    slow_turning_mb:=H_SlowTurning OR BR_ECR_PUBSH_ALARM_TEST;    (*PRORCCAN1001	  slow_turning_mb      %QX284.0*)

       slow_turnok_mb:=SLOWTURNOK;      (*PRORCCAN1002	  slow_turnok_mb	      %QX284.1*)

       slow_turning_failure_mb:=SlowTurningFailure OR BR_ECR_PUBSH_ALARM_TEST ; (*PRORCCAN1003	low_turning_failure_mb	%QX284.2*)

	start_failure_alm:=startFail OR BR_ECR_PUBSH_ALARM_TEST;(*PRORCCAN1004   start_failure_alm   	%QX284.3*)

     start_air_valve_man_closed:=StartAirValueManClosedBX  OR BR_ECR_PUBSH_ALARM_TEST ;	(*PRORCCAN1005	start_air_valve_man_closed     %QX284.4*)

      turning_gear_engaged_alm:=H_TurnGearEngaged OR BR_ECR_PUBSH_ALARM_TEST;           (*PRORCCAN1006	turning_gear_engaged_alm	    %QX284.5-------------------------------------------*)

       turning_gear_sensor_failure_alm:=H_TurnGearSensorFail OR BR_ECR_PUBSH_ALARM_TEST;  (*PRORCCAN1007	turning_gear_sensor_failure_alm	%QX284.6 *)

       any_aux_blower_run_mb:=AnyAuxBlowerRun  OR BR_ECR_PUBSH_ALARM_TEST ;         (*PRORCCAN1008 	any_aux_blower_run_mb	      %QX284.7*)

       aux_blower_manctrl_mb:=H_AuxBlowerManCTRL;(*PRORCCAN1009	aux_blower_manctrl_mb  	%QX284.8*)

       aux_blower_failed_mb:=H_AuxBlowerFailed OR BR_ECR_PUBSH_ALARM_TEST;           (*PRORCCAN1010	aux_blower_failed_mb	       %QX284.9*)

       speed_prgm_override:=H_SPD_PRGM_OVERD;    (* PRORCCAN1011	speed_prgm_override   	       %QX284.10*)

       eng_output_limited:=H_ENG_OUTPUT_LIMITED;   (*PRORCCAN1012	eng_output_limited            	%QX284.11*)

       setpoint_critical_speed:=H_SETPOINT_CRITICAL_SPD_BX; (*PRORCCAN1013	setpoint_critical_speed    	%QX284.12 *)

       eng_critical_speed:=H_ENG_CRITICAL_SPD_BX;   (*PRORCCAN1014	eng_critical_speed     	%QX284.13*)

	unic_start_learning_inprogress_indica:= H_StartLearningInPro OR BR_ECR_PUBSH_ALARM_TEST; (*PRORCCAN1015	unic_start_learning_inprogress_indica  	%QX284.14*)

       speed_prgm_active:=H_SPEED_PRGM_ACTIVE;(*PRORCCAN1016   speed_prgm_active    %QX284.15*)

       bridge_ctrl:=BR_CTRL;(* PRORCCAN2001 	bridge_ctrl  	%QX285.0*)

        ecr_aut_ctrl:=ECRA_CTRL;  (*PRORCCAN2002	ecr_aut_ctrl  	%QX285.1*)

	 ecr_man_ctrl:=ECRM_CTRL;(*PRORCCAN2003	ecr_man_ctrl  	%QX285.2*)

	 local_man_ctrl:=LOC_MAN_CTRL;(*PRORCCAN2004 	local_man_ctrl  	%QX285.3*)

       br_lamp_br_flash:=BRG_BRG_CTRL_FLSH;      (*PRORCCAN2005	br_lamp_br_flash  	%QX285.4*)

	br_lamp_ecr_autom_flash:=BRG_ECRA_CTRL_FLSH;    (*PRORCCAN2006	br_lamp_ecr_autom_flash  	%QX285.5*)

	br_lamp_ecr_man_flash:=BRG_ECRM_CTRL_FLSH;   (*PRORCCAN2007	br_lamp_ecr_man_flash  	%QX285.6*)

	br_lamp_local_man_flash:=BRG_LOCAL_MAN_CTRL_FLSH;     (*PRORCCAN2008	br_lamp_local_man_flash  	%QX285.7*)

	br_accoustic_ctrl_transfer_signal:= BR_ACCOUST_CTRL_SIGN_BX;  (*PRORCCAN2009	br_accoustic_ctrl_transfer_signal  	%QX285.8*)

	ecr_lamp_br_flash:=ECR_BRG_CTRL_FLSH;   (*PRORCCAN2010	ecr_lamp_br_flash  	%QX285.9*)

	 ecr_lamp_ecr_autom_flash:=ECR_ECRA_CTRL_FLSH;(*PRORCCAN2011	ecr_lamp_ecr_autom_flash  	%QX285.10*)

	ecr_lamp_ecr_man_flash:=ECR_ECRM_CTRL_FLSH;(*PRORCCAN2012	ecr_lamp_ecr_man_flash   	%QX285.11*)

	ecr_lamp_local_man_flash:=ECR_LOCAL_MAN_CTRL_FLSH  ;(*PRORCCAN2013	ecr_lamp_local_man_flash   	%QX285.12*)

	ecr_ccoustic_ctrl_transfer_signal:= ECR_ACCOUST_CTRL_SIGN_BX ;  (*PRORCCAN2014	ecr_ccoustic_ctrl_transfer_signal  	%QX285.13*)

       shaft_locking_dev_engaged:= H_ShtLockDevEngaged OR BR_ECR_PUBSH_ALARM_TEST; (*PRORCCAN2015	  shaft_locking_dev_engaged     %QX285.14*)

       over_speed_rcs_mb:=OVER_SPEED;(*PRORCS0001   over_speed_rcs_mb	%QX286.0*)

	rcs_overspeed_sw:=RCS_SW_overspd;(*PRORCS0047	rcs_overspeed_sw  	%QX286.1*)

	rcs_overspeed_hw_mb:= RCS_HW_overspd; (*PRORCS0048	rcs_overspeed_hw_mb  	%QX286.2 *)

	air_run_indicator:=H_AIRRUN_BR_ECR;(*PRORCS0049	air_run_indicator  	%QX286.3*)

      rcs_mvl_br_failure:=MVL_BR_FAIL;(*PRORCS0050	rcs_mvl_br_failure  	%QX286.4*)

	rcs_mvl_ecr_failure:=MVL_ECR_FAIL;(*PRORCS0051	rcs_mvl_ecr_failure  	%QX286.5*)

       aux_blower_preselecRC_mb:=H_AuxBlowerPresel;(*PRORCS0052	aux_blower_preselecRC_mb	%QX286.6*)

	chief_limit_speed_indicaotr:=HMI_BR_ECRA_CHIEFLIMIT;  (*PRORCS0057	chief_limit_speed_indicaotr  	%QX286.7*)

       rcs_eng_speed_sensor1_failure:=RCS_SPD_SENSOR_FAIL1 OR BR_ECR_PUBSH_ALARM_TEST;    (*PRORCS0058	rcs_eng_speed_sensor1_failure	%QX286.8*)

	rcs_eng_speed_sensor2_failure:=RCS_SPD_SENSOR_FAIL2 OR BR_ECR_PUBSH_ALARM_TEST;  (*PRORCS0059	rcs_eng_speed_sensor2_failure	%QX286.9 *)

        startair_press_low_alm:=H_StartAirPressLow  OR BR_ECR_PUBSH_ALARM_TEST;  (*PRORCS0063	startair_press_low_alm   	%QX286.10----*)

       start_interlock_alm:= H_StartInterlock OR BR_ECR_PUBSH_ALARM_TEST 	;(*PRORCS0064	start_interlock_alm  	%QX286.11*)

       propulsion_ctrl_failure_alm_mb:=propulsion_ctrl_failure_alm;  (*PRORCS0069 	propulsion_ctrl_failure_alm   	%QX286.12*)

       propulsion_ctrl_passive_failure_alm_mb:=propulsion_ctrl_passive_failure_alm;(*  PRORCS0070  propulsion_ctrl_passive_failure_alm_mb  %QX286.13*)

	propulsion_ctrl_speed_meas_failure_alm:=PCS_SPD_MEASURE_FAILURE; (*PRORCS0071	propulsion_ctrl_speed_meas_failure_alm  	%QX286.14*)

       rcs_comm_to_unic_lost_failure:=CommunicationLost OR BR_ECR_PUBSH_ALARM_TEST;	(* PRORCS0072	rcs_comm_to_unic_lost_failure  	%QX287.0*)

       rcs_can1_TO_unic_lost_failure:=BreakDownCAN1 OR  BR_ECR_PUBSH_ALARM_TEST;	(*PRORCS0073	rcs_can1_TO_unic_lost_failure  	%QX287.1*)

       rcs_can2_to_unic_lost_failure:=BreakDownCAN2 OR  BR_ECR_PUBSH_ALARM_TEST ;  	(*PRORCS0074	rcs_can2_TO_unic_lost_failure  	%QX287.2*)

	eng_starting:= START AND (EngTurnINCRSPDir AND  NOT EngineStandstill )  OR BR_ECR_PUBSH_ALARM_TEST; (*PRORCS0075	eng_starting  	%QX287.3*)

	eng_running:=EngineRun OR BR_ECR_PUBSH_ALARM_TEST; (*PRORCS0076	eng_running  	%QX287.4*)

	eng_ready_for_start:= NOT  eng_not_ready OR BR_ECR_PUBSH_ALARM_TEST; (*PRORCS0077	eng_ready_for_start  	%QX287.5*)

	eng_not_ready:=StartInterlock  OR CommunicationLost  OR BR_ECR_PUBSH_ALARM_TEST ;(*PRORCS0078	eng_not_ready  	%QX287.6*)

	eng_stopping:=( NOT NNBrake AND  BRAKE  ) OR BR_ECR_PUBSH_ALARM_TEST; (*PRORCS0079 	eng_stopping  	%QX287.7*)

	eng_stopped:=EngineStandstill;(*PRORCS0080	eng_stopped  	%QX287.8*)

	rcs_eng_speed2:=ANALOG_DETECT_SPEED_RCS;(*PRORCS0081	rcs_eng_speed2	%QX300*)

	safety_system_off:= SafetySystemOff  OR BR_ECR_PUBSH_ALARM_TEST;  (*PRORCS0082	safety_system_off  	%QX287.10*)

	eng_tripped_mb:=eng_tripped OR BR_ECR_PUBSH_ALARM_TEST;   (*eng_tripped_mb  AT  %QX266.11:BOOL  ;*)(*PRORCS0083	eng_tripped  	%QX287.11*)

	mvl_postion_ahead  :=MVL_POS_AHD  ;(*PRORCS0091	mvl_postion_ahead  	%QX287.12*)

	mvl_postion_astern :=MVL_POS_AST ;(*PRORCS0092	mvl_postion_astern  	%QX287.13*)

	mvl_postion_stop  :=MVL_POS_STOP;(*PRORCS0093	mvl_postion_stop  	%QX287.14*)

	ahead_cmd:=AHEAD;   (*PRORCS0094	ahead_cmd  	%QX288.0*)

	 astern_cmd:=   ASTERN;    (*PRORCS0095	astern_cmd  	%QX288.1*)

	stop_cmd:=STOP;   (*PRORCS0096	stop_cmd  	%QX288.2*)

       rcs_eng_turning_ahead :=EngTurningAHD; (*PRORCS0099	rcs_eng_turning_ahead  	%QX288.3*)

	rcs_eng_turning_astern := EngTurningAST ; (*PRORCS0100	rcs_eng_turning_astern   	%QX288.4*)

       pcs_system_ready:= RemoteCtrl AND NOT (CommunicationLost  OR ess_can_communicationLost  OR  propulsion_ctrl_failure_alm OR  SafetySystemOff) OR BR_ECR_PUBSH_ALARM_TEST ;(*PRORCS0103	pcs_system_ready  	%QX288.5    ALARM  TEST*)

       plant_interlock:=PlantInterlock;(*PRORCS0107	plant_interlock  	%QX288.6*)

        remote_ctrl_failure:=propulsion_ctrl_failure_alm  OR BR_ECR_PUBSH_ALARM_TEST; (*PRORCS0108	remote_ctrl_failure  	%QX288.7 *)

	(* wrong_way_alm:=H_WRONG_WAY_ALARM;(*PRORCS0109	wrong_way_alm  	%QX288.8*)--------------DELETE*)

        ecr_lamp_test_pb_mb:=ECR_LAMP_TEST_PB_INTERNAL;(*PRORCS0139	ecr_lamp_test_pb_mb	%QX288.9*)

        br_lamp_test_pb_mb:=BR_LAMP_TEST_PB_INTERNAL;(*PRORCS0140	br_lamp_test_pb_mb	%QX288.10*)

	  br_portlamp_test_pb_mb:=BR_LAMP_TEST_PB_INTERNAL;(*PRORCS0141	br_portlamp_test_pb_mb	%QX288.11*)

	 br_stbdlamp_test_pb_mb:=BR_LAMP_TEST_PB_INTERNAL;(*PRORCS0142	br_stbdlamp_test_pb_mb	%QX288.12 *)

       spd_sim_mode_active_mb:=SPD_SIM_MODE_ACTIVE_FLAG;(* PRORCS0157	spd_sim_mode_active_mb	%QX289.11*)

	 startfail_horn_alm_mb:=Start_Fail_Flash_sign;   (*PRORCS0158   	StartFail HORN ALARM		SP_swd_perm_rcs6_13_62 	*)

      (* horn_alarm_mb:=(H_HORN_ALARM_ECR OR H_HORN_ALARM_BRG  OR ENG_FAIL_ACOUSTIC OR BR_ECR_PUBSH_ALARM_TEST) ; *)(*PRORCS0164	horn_alarm_mb	%QX289.13*)


        port_ctrl_rc_es:= PORT_CTRL_EOT ;(*PRORCS9001	port_ctrl_rc_es	%QX287.9*)

        stbd_ctrl_rc_es:=STBD_CTRL_EOT ;(*PRORCS9002	stbd   ctrl_rc_es*)

        rcs_speed_meansure_value_mb:=RCS_SPEED_MEANSURE_VALUE;(*PRORCS9003	rcs_speed_meansure_value_mb	%QX302*)

        safety_sys_stop_mb:=  SafetyStop;(*PRORCS9004*)

        br_mvl_level_mb:=BR_MVL_LEVEL;(*%QW370*)

        ecr_mvl_level_mb:=ECR_MVL_LEVEL;(*%QW372*)

       br_ecr_pubsh_alarm_test_mb:=BR_ECR_PUBSH_ALARM_TEST;

	h_br_mvl_rpm_cmd_mb:=BR_MVL_RPM_CMD ;(*%QW468*)

	h_ecr_mvl_rpm_cmd_mb:=MCR_MVL_RPM_CMD;(*%QW470*)
END_FUNCTION_BLOCK

(* POU Configuration/MODBUS_CONFIGURATION, ST *)
PROGRAM MODBUS_CONFIGURATION        
VAR                                
END_VAR                            
(*                                 
   <?xml version="1.0" encoding="UTF-16" standalone="yes"?>
<network xml_structure_version="1">
	<generator_settings minRTUTaskCycleTimeMs="5" minEthaskCycleTimeMs="5" ethSlaveMultiplier="0.1" rtuInterfaceMultiplier="0.1" taskGeneration="false"/>
	<master_interface type="eth" name="" expanded="true">
		<mb_slave comment="Ethernet MR Controller 100MBit 2Port" name="ESS" expanded="false" type="wago" article-no="0750-0882">
			<mb_connection type="eth" transport="UDP" port="502" ip="192.168.1.2" unitid="2" request_delay_ms="0" response_timeout_ms="50"/>
			<service_connection type="eth" ip="192.168.1.2"/>
			<generic_vars comment="" expanded="false"/>
			<pfc_vars comment="" expanded="true">
				<pfc_var name="ess_eng_turning_ahead_bkp_cfg" comment="" data_type="BOOL" iec_addr="%QX272.0" expanded="false" mb_access="ro" explicitAccess="false"/>
				<pfc_var name="ess_eng_turning_astern_bkp_cfg" comment="" data_type="BOOL" iec_addr="%QX272.1" expanded="false" mb_access="ro" explicitAccess="false"/>
				<pfc_var name="ess_eng_standstill_bkp_cfg" comment="" data_type="BOOL" iec_addr="%QX270.0" expanded="false" mb_access="ro" explicitAccess="false"/>
				<pfc_var name="ess_overspeed_sw_bkp_cfg" comment="" data_type="BOOL" iec_addr="%QX271.11" expanded="false" mb_access="ro" explicitAccess="false"/>
				<pfc_var name="ess_overspeed_hw_bkp_cfg" comment="" data_type="BOOL" iec_addr="%QX272.2" expanded="false" mb_access="ro" explicitAccess="false"/>
				<pfc_var name="alrm_acksound_off_br_cfg" comment="" data_type="BOOL" iec_addr="%QX274.1" expanded="false" mb_access="ro" explicitAccess="false"/>
				<pfc_var name="alrm_acksound_off_ecr_cfg" comment="" data_type="BOOL" iec_addr="%QX274.2" expanded="false" mb_access="ro" explicitAccess="false"/>
				<pfc_var name="alrm_acksound_off_port_cfg" comment="" data_type="BOOL" iec_addr="%QX274.3" expanded="false" mb_access="ro" explicitAccess="false"/>
				<pfc_var name="alrm_acksound_off_stbd_cfg" comment="" data_type="BOOL" iec_addr="%QX274.4" expanded="false" mb_access="ro" explicitAccess="false"/>
				<pfc_var name="safety_stop_cfg" comment="" data_type="BOOL" iec_addr="%QX271.13" expanded="false" mb_access="ro" explicitAccess="false"/>
				<pfc_var name="ess_eng_speed_bkp_cfg" comment="" data_type="REAL" iec_addr="%QW256" expanded="false" mb_access="ro" explicitAccess="false"/>
				<pfc_var name="ess_can_communicationLost_cfg" comment="" data_type="BOOL" iec_addr="%QX270.7" expanded="false" mb_access="ro" explicitAccess="false"/>
			</pfc_vars>
			<k_bus comment="" expanded="false"/>
		</mb_slave>
		<mb_slave comment="Ethernet MR Controller 100MBit 2Port" name="EOT" expanded="false" type="wago" article-no="0750-0882">
			<mb_connection type="eth" transport="UDP" port="502" ip="192.168.1.3" unitid="3" request_delay_ms="0" response_timeout_ms="50"/>
			<service_connection type="eth" ip="192.168.1.3"/>
			<generic_vars comment="" expanded="false"/>
			<pfc_vars comment="" expanded="true">
				<pfc_var name="BR_MVL_cfg" comment="" data_type="WORD" iec_addr="%QW0" expanded="false" mb_access="ro" explicitAccess="false"/>
				<pfc_var name="ECR_MVL_cfg" comment="" data_type="WORD" iec_addr="%QW1" expanded="false" mb_access="ro" explicitAccess="false"/>
			</pfc_vars>
			<k_bus comment="" expanded="false"/>
		</mb_slave>
		<mb_slave comment="Ethernet MR Controller 100MBit 2Port" name="ESS_2" expanded="true" type="wago" article-no="0750-0882">
			<mb_connection type="eth" transport="UDP" port="502" ip="192.168.2.2" unitid="2" request_delay_ms="0" response_timeout_ms="50"/>
			<service_connection type="eth" ip="192.168.1.2"/>
			<generic_vars comment="" expanded="false"/>
			<pfc_vars comment="" expanded="true">
				<pfc_var name="ess_eng_turning_ahead_bkp_cfg" comment="" data_type="BOOL" iec_addr="%QX272.0" expanded="false" mb_access="ro" explicitAccess="false"/>
				<pfc_var name="ess_eng_turning_astern_bkp_cfg" comment="" data_type="BOOL" iec_addr="%QX272.1" expanded="false" mb_access="ro" explicitAccess="false"/>
				<pfc_var name="ess_eng_standstill_bkp_cfg" comment="" data_type="BOOL" iec_addr="%QX270.0" expanded="false" mb_access="ro" explicitAccess="false"/>
				<pfc_var name="ess_overspeed_sw_bkp_cfg" comment="" data_type="BOOL" iec_addr="%QX271.11" expanded="false" mb_access="ro" explicitAccess="false"/>
				<pfc_var name="ess_overspeed_hw_bkp_cfg" comment="" data_type="BOOL" iec_addr="%QX272.2" expanded="false" mb_access="ro" explicitAccess="false"/>
				<pfc_var name="alrm_acksound_off_br_cfg" comment="" data_type="BOOL" iec_addr="%QX274.1" expanded="false" mb_access="ro" explicitAccess="false"/>
				<pfc_var name="alrm_acksound_off_ecr_cfg" comment="" data_type="BOOL" iec_addr="%QX274.2" expanded="false" mb_access="ro" explicitAccess="false"/>
				<pfc_var name="alrm_acksound_off_port_cfg" comment="" data_type="BOOL" iec_addr="%QX274.3" expanded="false" mb_access="ro" explicitAccess="false"/>
				<pfc_var name="alrm_acksound_off_stbd_cfg" comment="" data_type="BOOL" iec_addr="%QX274.4" expanded="false" mb_access="ro" explicitAccess="false"/>
				<pfc_var name="safety_stop_cfg" comment="" data_type="BOOL" iec_addr="%QX271.13" expanded="false" mb_access="ro" explicitAccess="false"/>
				<pfc_var name="ess_eng_speed_bkp_cfg" comment="" data_type="REAL" iec_addr="%QW256" expanded="false" mb_access="ro" explicitAccess="false"/>
				<pfc_var name="ess_can_communicationLost_cfg" comment="" data_type="BOOL" iec_addr="%QX270.7" expanded="false" mb_access="ro" explicitAccess="false"/>
			</pfc_vars>
			<k_bus comment="" expanded="false"/>
		</mb_slave>
	</master_interface>
</network>
                              
*)                                 
;                                  
END_PROGRAM

(* POU Generated Code/Ethernet/MBCFG_ESS, ST *)
PROGRAM MBCFG_ESS(* generated by config one prg for each slave *)

VAR_INPUT

END_VAR

VAR_OUTPUT
       ess_eng_turning_ahead_bkp_cfg       :    BOOL;       (**) 
       ess_eng_turning_astern_bkp_cfg       :    BOOL;       (**) 
       ess_eng_standstill_bkp_cfg       :    BOOL;       (**) 
       ess_overspeed_sw_bkp_cfg       :    BOOL;       (**) 
       ess_overspeed_hw_bkp_cfg       :    BOOL;       (**) 
       alrm_acksound_off_br_cfg       :    BOOL;       (**) 
       alrm_acksound_off_ecr_cfg       :    BOOL;       (**) 
       alrm_acksound_off_port_cfg       :    BOOL;       (**) 
       alrm_acksound_off_stbd_cfg       :    BOOL;       (**) 
       safety_stop_cfg       :    BOOL;       (**) 
       ess_eng_speed_bkp_cfg       :    REAL;       (**) 
       ess_can_communicationLost_cfg       :    BOOL;       (**) 

    (*--- system variables (read only) ----------------------------------------*)
    MBCFG_IpAddress :   STRING(11) := '192.168.1.2'; (* address of this slave *)
    MBCFG_Port      :   UINT := 502;
    MBCFG_UnitID    :   BYTE := 2;
    MBCFG_TimeOut   :   TIME := t#50ms;
    MBCFG_Error     :   MBCFG_eERROR;
    (*-------------------------------------------------------------------------*)
END_VAR

{library private}
VAR CONSTANT
    zz_VARIABLECOUNT:   INT := 12;	(* number of variables 	*)
    zz_JOBCOUNT     :   INT := 2; 	(* number of jobs		*)
END_VAR
VAR

    (*=== VARIABLE LIST ===============================================================================*)
    zz_VariableList :   ARRAY[1..zz_VARIABLECOUNT] OF MBCFG_typVARIABLE :=
    (   BitSize         := 1,
        ptVar           := 0,
        ReadJobIndex    := 1,
        ReadStartBitNo  := 32,
        WriteJobIndex   := 0,
        WriteStartBitNo := 0 ),
    (   BitSize         := 1,
        ptVar           := 0,
        ReadJobIndex    := 1,
        ReadStartBitNo  := 33,
        WriteJobIndex   := 0,
        WriteStartBitNo := 0 ),
    (   BitSize         := 1,
        ptVar           := 0,
        ReadJobIndex    := 1,
        ReadStartBitNo  := 0,
        WriteJobIndex   := 0,
        WriteStartBitNo := 0 ),
    (   BitSize         := 1,
        ptVar           := 0,
        ReadJobIndex    := 1,
        ReadStartBitNo  := 27,
        WriteJobIndex   := 0,
        WriteStartBitNo := 0 ),
    (   BitSize         := 1,
        ptVar           := 0,
        ReadJobIndex    := 1,
        ReadStartBitNo  := 34,
        WriteJobIndex   := 0,
        WriteStartBitNo := 0 ),
    (   BitSize         := 1,
        ptVar           := 0,
        ReadJobIndex    := 1,
        ReadStartBitNo  := 65,
        WriteJobIndex   := 0,
        WriteStartBitNo := 0 ),
    (   BitSize         := 1,
        ptVar           := 0,
        ReadJobIndex    := 1,
        ReadStartBitNo  := 66,
        WriteJobIndex   := 0,
        WriteStartBitNo := 0 ),
    (   BitSize         := 1,
        ptVar           := 0,
        ReadJobIndex    := 1,
        ReadStartBitNo  := 67,
        WriteJobIndex   := 0,
        WriteStartBitNo := 0 ),
    (   BitSize         := 1,
        ptVar           := 0,
        ReadJobIndex    := 1,
        ReadStartBitNo  := 68,
        WriteJobIndex   := 0,
        WriteStartBitNo := 0 ),
    (   BitSize         := 1,
        ptVar           := 0,
        ReadJobIndex    := 1,
        ReadStartBitNo  := 29,
        WriteJobIndex   := 0,
        WriteStartBitNo := 0 ),
    (   BitSize         := 32,
        ptVar           := 0,
        ReadJobIndex    := 2,
        ReadStartBitNo  := 0,
        WriteJobIndex   := 0,
        WriteStartBitNo := 0 ),
    (   BitSize         := 1,
        ptVar           := 0,
        ReadJobIndex    := 1,
        ReadStartBitNo  := 7,
        WriteJobIndex   := 0,
        WriteStartBitNo := 0 )

                        ;
    (*=================================================================================================*)

    (*=== JOB LIST ====================================================================================*)
    zz_JobList     :   ARRAY[1..zz_JOBCOUNT] OF MBCFG_typCOM_JOB :=
     (   Functioncode            := 2,
        ReadStartAddress        := 4320,
        ReadQuantity            := 69,
        WriteStartAddress       := 0,
        WriteQuantity           := 0,
        ptReadData              := 0, 
        ptWriteData             := 0 ),
     (   Functioncode            := 4,
        ReadStartAddress        := 256,
        ReadQuantity            := 2,
        WriteStartAddress       := 0,
        WriteQuantity           := 0,
        ptReadData              := 0, 
        ptWriteData             := 0 )

                        ;
    (*=================================================================================================*)

    (*=== DATA FIELDS =================================================================================*)
     zz_DataField_1_Read       :       ARRAY[1..5] OF WORD;
     zz_DataField_2_Read       :       ARRAY[1..2] OF WORD;
	
    (*=================================================================================================*)

    (*=== MODBUS MASTER =====================================*)
    zz_MBCFG_MASTER_ETH :       MBCFG_MASTER_UDP;
    (*=======================================================*)

END_VAR
(*--- for each variable -------------------------*)
   zz_VariableList[1].ptVar := ADR(ess_eng_turning_ahead_bkp_cfg);
   zz_VariableList[2].ptVar := ADR(ess_eng_turning_astern_bkp_cfg);
   zz_VariableList[3].ptVar := ADR(ess_eng_standstill_bkp_cfg);
   zz_VariableList[4].ptVar := ADR(ess_overspeed_sw_bkp_cfg);
   zz_VariableList[5].ptVar := ADR(ess_overspeed_hw_bkp_cfg);
   zz_VariableList[6].ptVar := ADR(alrm_acksound_off_br_cfg);
   zz_VariableList[7].ptVar := ADR(alrm_acksound_off_ecr_cfg);
   zz_VariableList[8].ptVar := ADR(alrm_acksound_off_port_cfg);
   zz_VariableList[9].ptVar := ADR(alrm_acksound_off_stbd_cfg);
   zz_VariableList[10].ptVar := ADR(safety_stop_cfg);
   zz_VariableList[11].ptVar := ADR(ess_eng_speed_bkp_cfg);
   zz_VariableList[12].ptVar := ADR(ess_can_communicationLost_cfg);

(*-----------------------------------------------*)

(*--- for each job -----------------------------------*)
zz_JobList[1].ptReadData   := ADR(zz_DataField_1_Read);
zz_JobList[2].ptReadData   := ADR(zz_DataField_2_Read);

(*----------------------------------------------------*)


(*#### START OF FIXED CODE #####################################*)
zz_MBCFG_MASTER_ETH(	strIpAddress    := MBCFG_IpAddress,
                        uiPort          := MBCFG_Port,
                        bUnitID         := MBCFG_UnitID,
                        tTimeOut        := MBCFG_TimeOut,
                        iVariableCount  := zz_VARIABLECOUNT,
                        ptVariableList  := ADR(zz_VariableList),
                        iJobCount       := zz_JOBCOUNT,
                        ptJobList       := ADR(zz_JobList),
                        eError          => MBCFG_Error
                    );
(*##############################################################*)
END_PROGRAM

(* POU Generated Code/Ethernet/MBCFG_ESS_2, ST *)
PROGRAM MBCFG_ESS_2(* generated by config one prg for each slave *)

VAR_INPUT

END_VAR

VAR_OUTPUT
       ess_eng_turning_ahead_bkp_cfg       :    BOOL;       (**) 
       ess_eng_turning_astern_bkp_cfg       :    BOOL;       (**) 
       ess_eng_standstill_bkp_cfg       :    BOOL;       (**) 
       ess_overspeed_sw_bkp_cfg       :    BOOL;       (**) 
       ess_overspeed_hw_bkp_cfg       :    BOOL;       (**) 
       alrm_acksound_off_br_cfg       :    BOOL;       (**) 
       alrm_acksound_off_ecr_cfg       :    BOOL;       (**) 
       alrm_acksound_off_port_cfg       :    BOOL;       (**) 
       alrm_acksound_off_stbd_cfg       :    BOOL;       (**) 
       safety_stop_cfg       :    BOOL;       (**) 
       ess_eng_speed_bkp_cfg       :    REAL;       (**) 
       ess_can_communicationLost_cfg       :    BOOL;       (**) 

    (*--- system variables (read only) ----------------------------------------*)
    MBCFG_IpAddress :   STRING(11) := '192.168.2.2'; (* address of this slave *)
    MBCFG_Port      :   UINT := 502;
    MBCFG_UnitID    :   BYTE := 2;
    MBCFG_TimeOut   :   TIME := t#50ms;
    MBCFG_Error     :   MBCFG_eERROR;
    (*-------------------------------------------------------------------------*)
END_VAR

{library private}
VAR CONSTANT
    zz_VARIABLECOUNT:   INT := 12;	(* number of variables 	*)
    zz_JOBCOUNT     :   INT := 2; 	(* number of jobs		*)
END_VAR
VAR

    (*=== VARIABLE LIST ===============================================================================*)
    zz_VariableList :   ARRAY[1..zz_VARIABLECOUNT] OF MBCFG_typVARIABLE :=
    (   BitSize         := 1,
        ptVar           := 0,
        ReadJobIndex    := 1,
        ReadStartBitNo  := 32,
        WriteJobIndex   := 0,
        WriteStartBitNo := 0 ),
    (   BitSize         := 1,
        ptVar           := 0,
        ReadJobIndex    := 1,
        ReadStartBitNo  := 33,
        WriteJobIndex   := 0,
        WriteStartBitNo := 0 ),
    (   BitSize         := 1,
        ptVar           := 0,
        ReadJobIndex    := 1,
        ReadStartBitNo  := 0,
        WriteJobIndex   := 0,
        WriteStartBitNo := 0 ),
    (   BitSize         := 1,
        ptVar           := 0,
        ReadJobIndex    := 1,
        ReadStartBitNo  := 27,
        WriteJobIndex   := 0,
        WriteStartBitNo := 0 ),
    (   BitSize         := 1,
        ptVar           := 0,
        ReadJobIndex    := 1,
        ReadStartBitNo  := 34,
        WriteJobIndex   := 0,
        WriteStartBitNo := 0 ),
    (   BitSize         := 1,
        ptVar           := 0,
        ReadJobIndex    := 1,
        ReadStartBitNo  := 65,
        WriteJobIndex   := 0,
        WriteStartBitNo := 0 ),
    (   BitSize         := 1,
        ptVar           := 0,
        ReadJobIndex    := 1,
        ReadStartBitNo  := 66,
        WriteJobIndex   := 0,
        WriteStartBitNo := 0 ),
    (   BitSize         := 1,
        ptVar           := 0,
        ReadJobIndex    := 1,
        ReadStartBitNo  := 67,
        WriteJobIndex   := 0,
        WriteStartBitNo := 0 ),
    (   BitSize         := 1,
        ptVar           := 0,
        ReadJobIndex    := 1,
        ReadStartBitNo  := 68,
        WriteJobIndex   := 0,
        WriteStartBitNo := 0 ),
    (   BitSize         := 1,
        ptVar           := 0,
        ReadJobIndex    := 1,
        ReadStartBitNo  := 29,
        WriteJobIndex   := 0,
        WriteStartBitNo := 0 ),
    (   BitSize         := 32,
        ptVar           := 0,
        ReadJobIndex    := 2,
        ReadStartBitNo  := 0,
        WriteJobIndex   := 0,
        WriteStartBitNo := 0 ),
    (   BitSize         := 1,
        ptVar           := 0,
        ReadJobIndex    := 1,
        ReadStartBitNo  := 7,
        WriteJobIndex   := 0,
        WriteStartBitNo := 0 )

                        ;
    (*=================================================================================================*)

    (*=== JOB LIST ====================================================================================*)
    zz_JobList     :   ARRAY[1..zz_JOBCOUNT] OF MBCFG_typCOM_JOB :=
     (   Functioncode            := 2,
        ReadStartAddress        := 4320,
        ReadQuantity            := 69,
        WriteStartAddress       := 0,
        WriteQuantity           := 0,
        ptReadData              := 0, 
        ptWriteData             := 0 ),
     (   Functioncode            := 4,
        ReadStartAddress        := 256,
        ReadQuantity            := 2,
        WriteStartAddress       := 0,
        WriteQuantity           := 0,
        ptReadData              := 0, 
        ptWriteData             := 0 )

                        ;
    (*=================================================================================================*)

    (*=== DATA FIELDS =================================================================================*)
     zz_DataField_1_Read       :       ARRAY[1..5] OF WORD;
     zz_DataField_2_Read       :       ARRAY[1..2] OF WORD;
	
    (*=================================================================================================*)

    (*=== MODBUS MASTER =====================================*)
    zz_MBCFG_MASTER_ETH :       MBCFG_MASTER_UDP;
    (*=======================================================*)

END_VAR
(*--- for each variable -------------------------*)
   zz_VariableList[1].ptVar := ADR(ess_eng_turning_ahead_bkp_cfg);
   zz_VariableList[2].ptVar := ADR(ess_eng_turning_astern_bkp_cfg);
   zz_VariableList[3].ptVar := ADR(ess_eng_standstill_bkp_cfg);
   zz_VariableList[4].ptVar := ADR(ess_overspeed_sw_bkp_cfg);
   zz_VariableList[5].ptVar := ADR(ess_overspeed_hw_bkp_cfg);
   zz_VariableList[6].ptVar := ADR(alrm_acksound_off_br_cfg);
   zz_VariableList[7].ptVar := ADR(alrm_acksound_off_ecr_cfg);
   zz_VariableList[8].ptVar := ADR(alrm_acksound_off_port_cfg);
   zz_VariableList[9].ptVar := ADR(alrm_acksound_off_stbd_cfg);
   zz_VariableList[10].ptVar := ADR(safety_stop_cfg);
   zz_VariableList[11].ptVar := ADR(ess_eng_speed_bkp_cfg);
   zz_VariableList[12].ptVar := ADR(ess_can_communicationLost_cfg);

(*-----------------------------------------------*)

(*--- for each job -----------------------------------*)
zz_JobList[1].ptReadData   := ADR(zz_DataField_1_Read);
zz_JobList[2].ptReadData   := ADR(zz_DataField_2_Read);

(*----------------------------------------------------*)


(*#### START OF FIXED CODE #####################################*)
zz_MBCFG_MASTER_ETH(	strIpAddress    := MBCFG_IpAddress,
                        uiPort          := MBCFG_Port,
                        bUnitID         := MBCFG_UnitID,
                        tTimeOut        := MBCFG_TimeOut,
                        iVariableCount  := zz_VARIABLECOUNT,
                        ptVariableList  := ADR(zz_VariableList),
                        iJobCount       := zz_JOBCOUNT,
                        ptJobList       := ADR(zz_JobList),
                        eError          => MBCFG_Error
                    );
(*##############################################################*)
END_PROGRAM

(* POU SWD, ST *)
FUNCTION_BLOCK SWD
VAR_INPUT
END_VAR
VAR_OUTPUT
END_VAR
VAR
	SRinst:SR;
	AIR_RUN_START_TEMP:BOOL;
	AIR_RUN_STOP_TEMP:BOOL;
	TOFInst_wgf: TOF;
	Slow_turning_staible:BOOL;
END_VAR
(*----------------SWD_swd_me_62   PROSWD0001----------------------*)
(*
IF   startFail   THEN   SWD_swd_me_62:=8;(*me_start_failure  8*)

ELSIF  ( NOT NNBrake)  AND  BRAKE    THEN  SWD_swd_me_62:=4 ;(* Stoping* ----------------ENG BRAKING???-------*)
(*ELSIF  (STOP AND EngineStandstill=FALSE)   THEN   SWD_swd_me_62:=4;(*me_stopping  4  *)*)
ELSIF   EngineRun    THEN   SWD_swd_me_62:=1;(* me_running    1 *)

ELSIF    EngineStandstill AND (NOT eng_ready_for_start)  THEN   SWD_swd_me_62:=3;(* me_stopped   3 *)
ELSIF    StartInterlock   THEN   SWD_swd_me_62:=2;(* me_startinterlock  2  *)
ELSIF   SlowTurningBX   THEN   SWD_swd_me_62:=6;(* me_slow_turning  6 *)
ELSIF   (PRESTART  AND   AnyAuxBlowerRun=FALSE)  THEN   SWD_swd_me_62:=7;(*PRESTART  7 *)
ELSIF   (EngTurnINCRSPDir AND START_BRAKE AND NOT  EngineStandstill ) THEN   SWD_swd_me_62:=5;(*me_starting  5 ----------------------STARTING  *)

ELSIF   EngTurnINCRSPDir AND NNstart AND (NOT PRESTART)  AND  (NOT  START)   THEN  SWD_swd_me_62:=18 ;(* SPD ACCELERATING*)

ELSIF   REVERSE_ACTIVE_SIGNAL  THEN  SWD_swd_me_62:=10;(*CRASH   ASTERN   10*)
ELSIF   SETPOINT_CRITICAL_SPD_BX   THEN  SWD_swd_me_62:=11;(*SETPOINT  CRITICAL  SPEED  11*)
ELSIF   SPEED_PRGM_ACTIVE_INDIC THEN  SWD_swd_me_62:=12;(*SPEED PROGRAM ACTIVE INDICATION   12*)
ELSIF   SPEED_OVERD_INDIC_BX    THEN  SWD_swd_me_62:=13;(*SPEED  PROGRAM  OVERRIDE  13*)
ELSIF   ENG_OUTPUT_LIMITED_BX     THEN  SWD_swd_me_62:=14;(*ENGINE OUTPUT LIMITED  14*)
ELSIF   ENG_CRITICAL_SPD_BX      THEN  SWD_swd_me_62:=15;(*ENGINE  CRITICAL SPEED   15*)
ELSIF   eng_ready_for_start     THEN  SWD_swd_me_62:=16 ;(* PRORCS0077 	ENGINE  READY  FOR  START    16 MODBUS SIGNAL*)
(*ELSIF  ( NOT NNBrake)  AND  BRAKE    THEN  SWD_swd_me_62:=17 ;(* speed decreasing*)*)

ELSE   SWD_swd_me_62:=0;(*me_unk 0*)
END_IF;
*)
IF   startFail   THEN   SWD_swd_me_62:=8;(*me_start_failure  8*)

ELSIF   BRAKE AND ( NOT NNBRAKE)     THEN  SWD_swd_me_62:=4 ;(* Stopping* ----------------ENG BRAKING???-------*)
(*ELSIF  (STOP AND EngineStandstill=FALSE)   THEN   SWD_swd_me_62:=4;(*me_stopping  4  *)*)
ELSIF   EngineRun   AND (NOT BRAKE) AND (NOT START) AND (NOT REVERSE_ACTIVE_SIGNAL)  THEN   SWD_swd_me_62:=1;(* me_running    1 *)

ELSIF    EngineStandstill AND (NOT eng_ready_for_start)  AND (NOT PRESTART) THEN   SWD_swd_me_62:=3;(* me_stopped   3 *)

ELSIF    StartInterlock  AND ( NOT eng_ready_for_start )   THEN   SWD_swd_me_62:=2;(* me_startinterlock  2  *)

(*ELSIF   SlowTurningBX   THEN   SWD_swd_me_62:=6;*)(* me_slow_turning  6 *)

ELSIF   PRESTART  AND (NOT START) THEN   SWD_swd_me_62:=7;(*PRESTART  7 *)

ELSIF  START AND (EngTurnINCRSPDir AND  NOT EngineStandstill )THEN   SWD_swd_me_62:=5;(*me_starting  5 ----------------------STARTING  *)

(*ELSIF   REVERSE_ACTIVE_SIGNAL  THEN  SWD_swd_me_62:=10;*)(*CRASH   ASTERN 10  no useful now --20170118*)
(*
ELSIF   SETPOINT_CRITICAL_SPD_BX  AND  (NOT StartInterlock ) THEN  SWD_swd_me_62:=11;(*SETPOINT  CRITICAL  SPEED  11*)

(*ELSIF   SPEED_PRGM_ACTIVE_INDIC THEN  SWD_swd_me_62:=12;*)(*SPEED PROGRAM ACTIVE INDICATION   12*)

ELSIF   SPEED_OVERD_INDIC_BX AND (NOT StartInterlock )   AND (NOT REVERSE_ACTIVE_SIGNAL ) THEN  SWD_swd_me_62:=13;(*SPEED  PROGRAM  OVERRIDE  13*)

ELSIF   ENG_OUTPUT_LIMITED_BX     THEN  SWD_swd_me_62:=14;(*ENGINE OUTPUT LIMITED  14*)

ELSIF   ENG_CRITICAL_SPD_BX      THEN  SWD_swd_me_62:=15;(*ENGINE  CRITICAL SPEED   15*)
*)
ELSIF   eng_ready_for_start  AND (NOT EngineRun) THEN  SWD_swd_me_62:=16 ;(* PRORCS0077 	ENGINE  READY  FOR  START    16 MODBUS SIGNAL*)

ELSE   SWD_swd_me_62:=0;(*me_unk 0*)
END_IF;

IF   SETPOINT_CRITICAL_SPD_BX  THEN  SWD_swd_merpmlim_0:=5;(*SETPOINT  CRITICAL  SPEED  5*)

ELSIF   SPEED_OVERD_INDIC_BX THEN  SWD_swd_merpmlim_0:=3;(*SPEED  PROGRAM  OVERRIDE  3*)

ELSIF   ENG_OUTPUT_LIMITED_BX     THEN  SWD_swd_merpmlim_0:=4;(*ENGINE OUTPUT LIMITED  4*)

ELSIF   ENG_CRITICAL_SPD_BX      THEN  SWD_swd_merpmlim_0:=6;(*ENGINE  CRITICAL SPEED   6*)

ELSIF   StartLearningInPro     THEN  SWD_swd_merpmlim_0:=7;(* START LEARNG IN PROGRESS 7*)

ELSIF   SPEED_PRGM_ACTIVE_INDIC      THEN  SWD_swd_merpmlim_0:=2;(* SPEED PROGRAM ACTIVE INDICATION 2*)

ELSE SWD_swd_merpmlim_0:=0;

END_IF

(*-----------------SWD_swd_cont_position_0   PROSWD0004---------------*)
IF            BR_CTRL        THEN SWD_swd_cont_position_0:=1;(*bridge_auto 1*)
ELSIF    ECRA_CTRL   THEN SWD_swd_cont_position_0:=2;(*mcr_auto 2  *)
ELSIF    ECRM_CTRL   THEN SWD_swd_cont_position_0:=3;(*mcr_man 3*)
ELSIF    LOC_MAN_CTRL     THEN SWD_swd_cont_position_0:=4;(*lop_man 4*)
ELSIF    PORT_CTRL_EOT   THEN SWD_swd_cont_position_0:=5;(*PORT WING 5*)
ELSIF    STBD_CTRL_EOT    THEN SWD_swd_cont_position_0:=6;(*STBD WING 6*)
ELSE     SWD_swd_cont_position_0:=0;(*ctr_pst_unk 0*)
END_IF;
(*----------------------------SWD_swd_mvl_direct_0---------------------*)
IF           MVL_POS_STOP     THEN       SWD_swd_mvl_direct_0:=3;(*mvl_direct_stop 3*)
ELSIF    MVL_POS_AHD       THEN       SWD_swd_mvl_direct_0:=1;(*mvl_direct_ahd 1*)
ELSIF    MVL_POS_AST        THEN       SWD_swd_mvl_direct_0:=2;(*mvl_direct_ast 2 *)
ELSE    SWD_swd_mvl_direct_0:=0;(* mvl_direct_unk 0*)
END_IF;

(*SWD_swd_aux_blower_62*)
IF             AuxBlowerFailed         THEN       SWD_swd_aux_blower_62:=3;(* aux_blower_fail 3*)
ELSIF     AnyAuxBlowerRun      THEN       SWD_swd_aux_blower_62:=1;(*aux_blower_running 1*)
ELSIF    AuxBlowerStop_PB      THEN       SWD_swd_aux_blower_62:=2;(*aux_blower_stopped 2*)
ELSIF    AuxBlowerManCTRL         THEN       SWD_swd_aux_blower_62:=4;(*aux_blower_man 4*)
ELSIF    AuxBlowerReselECRA_PB         THEN       SWD_swd_aux_blower_62:=5;(*aux_blowe Preselected 5--------------------------------------------TBD*)

ELSE     SWD_swd_aux_blower_62:=0;(* aux_blower_unk 0*)
END_IF;

(* SCS_swd_aux_blower_1_62    aux_blower_Preselect *)
IF          RemoteCtrl  OR AuxBlowerManCTRL      THEN  SCS_swd_aux_blower_1_62:=2;(*ALLOWED  2*)
ELSE  SCS_swd_aux_blower_1_62:=0;(*UNKNOWN    0*)
(*ELSIF  (NOT   AuxBlower_preslct_rc_ready)     THEN       SCS_swd_aux_blower_1_62:=3;(*ACTUAL_STATE_NOT_ALLOWED  3*)
ELSIF               AuxBlower_preslct_rc_ready      THEN       SCS_swd_aux_blower_1_62:=4;(* ACTUAL_STATE_ALLOWED   4*)
ELSIF ( NOT   AuxBlowerPreselectedRC)         THEN       SCS_swd_aux_blower_1_62:=5;(* IN_PROGRESS_NOT_ALLOWED  5*)
ELSIF              AuxBlowerPreselectedRC           THEN       SCS_swd_aux_blower_1_62:=6;(*IN_PROGRESS_ALLOWED  6*)
ELSE               SCS_swd_aux_blower_1_62:=0;  (*UNKNOWN    0*)*)
END_IF;
 (* SCS_swd_aux_blower_2_62    aux_blower_stopped*)
IF      RemoteCtrl  OR AuxBlowerManCTRL         THEN     SCS_swd_aux_blower_2_62:=2;(*ALLOWED  2*)
ELSE SCS_swd_aux_blower_2_62:=0;(*UNKNOWN    0*)
(*ELSIF          (NOT  AuxBlowerStop_PB   )                            THEN       SCS_swd_aux_blower_2_62:=3;(*ACTUAL_STATE_NOT_ALLOWED  3*)
ELSIF  (  AuxBlowerStop_PB   AND ECRA_CTRL)    THEN       SCS_swd_aux_blower_2_62:=4;(* ACTUAL_STATE_ALLOWED   4*)
ELSIF   ( NOT   AuxBlowerPreselectedRC)       THEN       SCS_swd_aux_blower_2_62:=6;(*IN_PROGRESS_ALLOWED  6*)
ELSE     SCS_swd_aux_blower_2_62:=0; (*UNKNOWN    0*)*)
END_IF;

(*SC_swd_aux_blower_62   aux_blower_running:=1,  aux_blower_stopped=2*)
IF          SC_swd_aux_blower_62=1     THEN   AuxBlowerReselECRA_PB:=TRUE ;
ELSIF   SC_swd_aux_blower_62=2   THEN  AuxBlowerStop_PB:=TRUE   ;
ELSE    AuxBlowerReselECRA_PB:=FALSE;    AuxBlowerStop_PB:=FALSE   ;
END_IF;


   (*SWD_swd_slow_turn_62 AT %QW279: UINT;*)
TOFInst_wgf(IN:=SlowTurningBX,PT:=T#0.5S);
Slow_turning_staible:=TOFInst_wgf.Q;
IF           SlowTurningFailure      THEN  SWD_swd_slow_turn_62:=3;(*slow_turn_fail *)
ELSIF   SlowTurnBRPush THEN  SWD_swd_slow_turn_62:=2;(*slow_turn_off*)
ELSIF      Slow_turning_staible    THEN  SWD_swd_slow_turn_62:=1;(*slow_turn_on 1*)
ELSIF    SLOWTURNOK            THEN  SWD_swd_slow_turn_62:=4;(*slow_trun_ok *)
ELSIF    SlowTurnQuest                 THEN  SWD_swd_slow_turn_62:=5;(*slow_turn_request *)
ELSIF    H_SlowTurnFailReset      THEN  SWD_swd_slow_turn_62:=6;(*slow_turn_reset *)
ELSE     SWD_swd_slow_turn_62:=0;(* slow_turning_unk*)
END_IF;

   (*SCS_swd_slow_turn_1_62   slow_turn_on 1*)
IF   RemoteCtrl OR  aheadastern     THEN  SCS_swd_slow_turn_1_62:=2;(*2  ALLOWED 2  *)
ELSIF (NOT RemoteCtrl)    THEN  SCS_swd_slow_turn_1_62:=0;(* UNKNOWN  0*)
(*ELSIF     STARTINTERLOCK        THEN  SCS_swd_slow_turn_1_62:=3;(*3 ACTUAL_STATE_NOT_ALLOWE 3*)
ELSIF        SlowTurnRCBX               THEN  SCS_swd_slow_turn_1_62:=4;(*ACTUAL_STATE_ALLOWED  4*)
ELSIF        STARTINTERLOCK        THEN  SCS_swd_slow_turn_1_62:=5;(*IN_PROGRESS_NOT_ALLOWED  5*)
ELSIF        NOT SLOWTURNOK     THEN  SCS_swd_slow_turn_1_62:=6;(* IN_PROGRESS_ALLOWED 6*)*)
END_IF;

   (*SCS_swd_slow_turn_6_62    slow_turn_reset 6*)
IF    (SlowTurnRCBX OR SlowTurningFailure)     THEN  SCS_swd_slow_turn_6_62:=2;(*2  ALLOWED 2  *)
ELSIF (NOT RemoteCtrl)   THEN  SCS_swd_slow_turn_6_62:=0;(* UNKNOWN  0*)
 (*ELSIF   (NOT H_SlowTurnFailReset )   THEN  SCS_swd_slow_turn_6_62:=3;(*3 ACTUAL_STATE_NOT_ALLOWE 3*)
ELSIF    H_SlowTurnFailReset                THEN  SCS_swd_slow_turn_6_62:=4;(*ACTUAL_STATE_ALLOWED  4*)
ELSIF    ( H_SlowTurnFailReset  AND   SlowTurningFailure  )   THEN  SCS_swd_slow_turn_6_62:=6;(* IN_PROGRESS_ALLOWED 6*)
ELSE    SCS_swd_slow_turn_6_62:=0;(*UNKNOWN  0*)*)
END_IF;

  (*SC_swd_slow_turn_62    slow_turn_on 1 *)
IF      SC_swd_slow_turn_62=1      AND BR_CTRL        THEN  SlowTurnBRPush:=TRUE;
ELSIF  SC_swd_slow_turn_62=1  AND ECRA_CTRL   THEN  SlowTurnECRAPush:=TRUE;
ELSE  SlowTurnBRPush:=FALSE;       SlowTurnECRAPush:=FALSE;
END_IF;
   (*SC_swd_slow_turn_62    slow_turn_reset 6  ;*)
IF          SC_swd_slow_turn_62=6 AND    BR_CTRL       THEN  SlowTurnFailReset_BR_PU:=TRUE;
ELSIF  SC_swd_slow_turn_62=6  AND   ECRA_CTRL  THEN  SlowTurnFailReset_ECRA_PU :=TRUE;
ELSE  SlowTurnFailReset_BR_PU:=FALSE;       SlowTurnFailReset_ECRA_PU:=FALSE;
END_IF;


(*---------------*)
 (*  SWD_swd_air_run_62    PROSWD0019 *)
IF         H_AIRRUN_BR_ECR(*  AIRRUN_RC_BX *)             THEN  SWD_swd_air_run_62:=1;(*air_run_on*)
ELSIF (NOT H_AIRRUN_BR_ECR )   THEN  SWD_swd_air_run_62:=2;(*air_run_off*)
ELSE  SWD_swd_air_run_62:=0;(*air_run_unk *)
END_IF;

  (* SC_swd_air_run_62      air_run_on  0/1    *)
(*
	IF  ( SC_swd_air_run_62=1 AND ECRA_CTRL) THEN
*)
      IF (CP_BUTAIRRUN>0.5 AND ECRA_CTRL) THEN

	 AIR_RUN_START_TEMP  :=TRUE;
	ELSE  AIR_RUN_START_TEMP :=FALSE;
	END_IF;
(*	IF  ( SC_swd_air_run_62=2 AND ECRA_CTRL) THEN
*)
      IF (CP_BUTAIRRUN<0.5 AND ECRA_CTRL) THEN

	 AIR_RUN_STOP_TEMP  :=TRUE;
	ELSE  AIR_RUN_STOP_TEMP :=FALSE;
	END_IF;
	SRinst (SET1:=AIR_RUN_START_TEMP , RESET:=AIR_RUN_STOP_TEMP);
	AIRRUN:=SRinst.Q1;

  (* SCS_swd_air_run_1_62            air_run_on*)
IF  ( ECRA_CTRL  AND(NOT  STARTINTERLOCK)  AND ( EngineStandstill OR  H_AIRRUN_BR_ECR  ) )THEN
(*SCS_swd_air_run_1_62:=2;(*2  ALLOWED 2 *)*)
PERAIRRUN:=TRUE;
ELSIF (NOT RemoteCtrl)    THEN
(*SCS_swd_air_run_1_62:=0;(*UNKNOWN  0*)*)
PERAIRRUN:=FALSE;
(*
ELSIF  STARTINTERLOCK   THEN  SCS_swd_air_run_1_62:=3;(*3 ACTUAL_STATE_NOT_ALLOWE 3*)
ELSIF  AIRRUN_RC_BX       THEN  SCS_swd_air_run_1_62:=4;(*ACTUAL_STATE_ALLOWED  4*)*)

END_IF;
END_FUNCTION_BLOCK

(* POU Critical_RPM, ST *)
FUNCTION_BLOCK Critical_RPM
VAR_INPUT
END_VAR
VAR_OUTPUT
END_VAR
VAR

END_VAR
IF  Critical_Speed_Enable =1
THEN
          IF SPEED_SETPOINT_BX> Critical_RPM_low1 AND SPEED_SETPOINT_BX<Critical_RPM_high1
          THEN SPEED_SETPOINT_BX:=Critical_RPM_low1;
          END_IF

ELSIF  Critical_Speed_Enable =2
THEN
          IF SPEED_SETPOINT_BX> Critical_RPM_low1 AND SPEED_SETPOINT_BX<Critical_RPM_high1
          THEN SPEED_SETPOINT_BX:=Critical_RPM_low1;
          END_IF

          IF SPEED_SETPOINT_BX> Critical_RPM_low2 AND SPEED_SETPOINT_BX<Critical_RPM_high2
          THEN SPEED_SETPOINT_BX:=Critical_RPM_low2;
          END_IF
END_IF
END_FUNCTION_BLOCK

(* POU Unic_Back, ST *)
FUNCTION_BLOCK Unic_Back
VAR_INPUT
END_VAR
VAR_OUTPUT
END_VAR
VAR
      FLASHER: BLINK;

	TON_INST: TON;
	TEMPOUT: BOOL;



	UNIC_RT: R_TRIG;
	A: BOOL;
END_VAR
IF  ENG_OUTPUT_LIMITED_BX
THEN
    (* FLASHER(ENABLE:=TRUE, TIMELOW:=T#500ms,TIMEHIGH:=T#500ms);
     OUTPUT_LIMIT_FLASHER:=FLASHER.OUT;*)
	OUTPUT_LIMIT_FLASHER:=FALSE;
ELSE
     OUTPUT_LIMIT_FLASHER:=FALSE;
END_IF;



IF  SPEED_PRGM_ACTIVE_INDIC
THEN
    (* FLASHER(ENABLE:=TRUE, TIMELOW:=T#500ms,TIMEHIGH:=T#500ms);
     SPEED_PRO_FLASHER:=FLASHER.OUT;*)
	SPEED_PRO_FLASHER:=FALSE;
ELSE
     SPEED_PRO_FLASHER:=FALSE;
END_IF;
END_FUNCTION_BLOCK

(* POU CANRead, ST *)
FUNCTION_BLOCK CANRead
VAR_INPUT
END_VAR
VAR_OUTPUT
END_VAR
VAR
	CANINOLD1: ARRAY [0..47] OF BYTE;
	CANINOLD2: ARRAY [0..47] OF BYTE;
	I: INT;
(*	CANIN1_CHG_FLAG:	BOOL;
	CANIN2_CHG_FLAG:	BOOL;*)

	CANIN_CHOICE:	BYTE;
       J: INT;

	POINT_ID: INT;
	TEMP: WORD;
END_VAR
(*figure  out  if  the CANIN1 and CANIN2 data are changing*)
FOR I:= 0	TO	 16	DO
	(*judge  CANIN1*)
	IF	BreakDownCAN1	=  FALSE
	THEN
		IF	CANIN1[10 + I] <> CANINOLD1[10 + I]
		THEN
			(*update  CANINOLD1 data*)
			CANINOLD1[10 + I] :=	CANIN1[10 + I];

			(*set CANIN1  change flag TRUE*)
			CANIN1_CHG_FLAG	:=  TRUE;
		END_IF
	END_IF

	(*judge  CANIN2*)
	IF	BreakDownCAN2	=  FALSE
	THEN
		IF	CANIN2[10 + I] <> CANINOLD2[10 + I]
		THEN
			(*update  CANINOLD2  data*)
			CANINOLD2[10 + I] :=	CANIN2[10 + I];

			(*set CANIN2  change flag TRUE*)
			CANIN2_CHG_FLAG	:=  TRUE;
		END_IF
	END_IF
END_FOR

(*如果CAN1和CAN2口数据同时改变，最终数据强制对应CAN1口，否则数据对应改变的CAN口*)
(*同时改变，数据强制对应CAN1口*)
IF	CANIN1_CHG_FLAG = TRUE  AND	CANIN2_CHG_FLAG = TRUE
THEN
	CANIN_CHOICE := 1;
(*CANIN1 数据发生变化，CANIN2数据未发生变化，数据对应CANIN1*)
ELSIF	CANIN1_CHG_FLAG	= TRUE  AND	CANIN2_CHG_FLAG	= FALSE
THEN
	CANIN_CHOICE := 1;
(*CANIN2 数据发生变化，CANIN1数据未发生变化，数据对应CANIN2*)
ELSIF	CANIN1_CHG_FLAG	= FALSE   AND    CANIN2_CHG_FLAG	= TRUE
THEN
	CANIN_CHOICE := 2;
ELSE
(*CANIN1,CANIN2数据均未发生变化*)
	CANIN_CHOICE  :=  0;
END_IF

CANIN1_CHG_FLAG	:=  FALSE;
CANIN2_CHG_FLAG	:=  FALSE;


(*choose CANIN1  data*)
IF	(CANIN_CHOICE  =  1 )
THEN
          FOR J:=0 TO 47 BY 1 DO
                ByteDataFromCAN[J]:=CANIN1[J];
          END_FOR;
END_IF


(*choose CANIN2  data*)
IF	CANIN_CHOICE  =  2
THEN
          FOR J:=0 TO 47 BY 1 DO
                ByteDataFromCAN[J]:=CANIN2[J];
          END_FOR;
END_IF

(*%QX48.2:=RecHeartBeatFLAG1;*)


(* Receive  Data  that   from CAN  store in DataFromCAN   (7~47)*)
POINT_ID:=ByteDataFromCAN[21]*256+ByteDataFromCAN[20];
IF(POINT_ID=2004)
THEN
 Estimated_Engine_Load_Internal :=  ByteDataFromCAN[25]*256+ByteDataFromCAN[24];
Fuel_Index_can := ByteDataFromCAN[23]*256+ByteDataFromCAN[22];
END_IF;

(*--------------------------------GET FROM CAN----------------------------- INPUT----------------------*)
(*ByteData[10]  ByteData[11]0X2002  start air pressure*)
 StartAirPressBX:=ByteDataFromCAN[11]*256+ByteDataFromCAN[10];

(*ByteDataFromCAN[12]   ByteDataFromCAN[13] UNIC INFO 0x2005 *)
SlowTurningBX:=ByteDataFromCAN[12].0;(*SLOWTURNING*)
SLOWTURNOK:=ByteDataFromCAN[12].1;(*SLOWTURNING OK*)
SlowTurnFailBX:= ByteDataFromCAN[12].2;(*SLOWTURNING FAILURE*)
Start_Failure_BX:=ByteDataFromCAN[12].3 ;(*START FAILURE *)
StartAirValueManClosedBX:=ByteDataFromCAN[12].4;(*START AIR VALVE MANUALLY CLOSED*)
TurningGearDiseng:= ByteDataFromCAN[12].5;(*TURNING GEAR  DISENGAGED *)
TurningGearSensorFail:=ByteDataFromCAN[12].6 ;(* TURNING GEAR SENSOR FAILURE*)
AnyAuxBlowerRun:= ByteDataFromCAN[12].7;(* ANY AUX.BLOWER RUNNING*)


AuxBlowerManCTRL:=ByteDataFromCAN[13].0 ; (* Set AUX.BLOWER MANUAL CONTROL*)
AuxBlowerFailed:=ByteDataFromCAN[13].1;(*ALL AUX. BLOWER FAILED *)
SPEED_OVERD_INDIC_BX:= ByteDataFromCAN[13].2 ;  (* SPEED PROGRAM OVERRIDE INDICATION*)
ENG_OUTPUT_LIMITED_BX:=ByteDataFromCAN[13].3;(*ENGINE OUTPUT LIMITED *)
SETPOINT_CRITICAL_SPD_BX:= ByteDataFromCAN[13].4; (* SETPOINT CRITICAL SPEED*)
ENG_CRITICAL_SPD_BX:= ByteDataFromCAN[13].5;  (*ENGINE CRITICAL SPEED *)
StartLearningInPro:= ByteDataFromCAN[13].6;(* START LEARNG IN PROGRESS*)
SPEED_PRGM_ACTIVE_INDIC:= ByteDataFromCAN[13].7;(* SPEED PROGRAM ACTIVE INDICATION *)



(*ByteDataFromCAN[14]   ByteDataFromCAN[15] 0x2006 control Tranfer feedback *)
BR_CTRL:=ByteDataFromCAN[14].0 ;(* BRIDGE CONTROL  2001*)
ECRA_CTRL:=ByteDataFromCAN[14].1;(*MCR AUTOM. CONTROL   2002*)
ECRM_CTRL:= ByteDataFromCAN[14].2;(*MCR MAN. CONTROL 2003 *)
LOC_MAN_CTRL:= ByteDataFromCAN[14].3;(*LOCAL MAN.CONTROL  2004*)
BRG_BRG_CTRL_FLSH:=ByteDataFromCAN[14].4;  (*BRIDGE LAMP "BRIDGE" FLASH  2005*)
BRG_ECRA_CTRL_FLSH:=  ByteDataFromCAN[14].5; (*BRIDGE LAMP "MCR AUTOM" FLASH  2006*)
BRG_ECRM_CTRL_FLSH:=ByteDataFromCAN[14].6; (*BRIDGE LAMP "MCR MAN" FLASH  2007*)
BRG_LOCAL_MAN_CTRL_FLSH := ByteDataFromCAN[14].7;(*BRIDGE LAMP "LOCAL MAN " FLASH  2008*)


H_HORN_ALARM_BRG:= ByteDataFromCAN[15].0;(*BRIDGE ACCOUSTIC CONTROL TRANSFER SIGNAL 2009*)
ECR_BRG_CTRL_FLSH:=ByteDataFromCAN[15].1;(*MCR LAMP "BRIDGE" FLASH *)
ECR_ECRA_CTRL_FLSH :=ByteDataFromCAN[15].2;(*MCR LAMP "MCR AUTOM" FLASH *)
ECR_ECRM_CTRL_FLSH :=ByteDataFromCAN[15].3;(*MCR LAMP "MCR MAN" FLASH *)
ECR_LOCAL_MAN_CTRL_FLSH :=ByteDataFromCAN[15].4;(*MCR LAMP "LOCAL  MAN" FLASH *)
H_HORN_ALARM_ECR:=ByteDataFromCAN[15].5;(*MCR ACCOUSTIC CONTROL TRANSFER SIGNAL *)
ShaftLockingDeviceEngaged:=  ByteDataFromCAN[15].6;(*SHAFT LOCKING DEVICE ENGAGED*)
END_FUNCTION_BLOCK

(* POU CANWrite, ST *)
FUNCTION_BLOCK CANWrite
VAR_INPUT
END_VAR
VAR_OUTPUT
END_VAR
VAR
	Temp_Word: WORD;

	CANOUT_OLD : ARRAY [0..47] OF BYTE;
	DATA_CHANGE_CAN1: BOOL;
	I :  BYTE;
END_VAR
(* -----------write data to CAN -------------------------OUTPUT-------------------------------------*)

(*--------- CANOUT1[10]   CANOUT1[11]  for  speed setpoint-----------*)

Temp_Word:=REAL_TO_WORD(SPEED_SETPOINT_BX*10);
CANOUT1[10]:=WORD_TO_BYTE(Temp_Word);
CANOUT1[11]:=WORD_TO_BYTE(SHR(Temp_Word ,8));

(*CANOUT[12]   CANOUT[13] store ENGINE COMMANDS   0X2003  *)
CANOUT1[12].0 := STOP ;(*STOP 0022*)
CANOUT1[12].1 :=START_BRAKE;(*START BREAK 0016*)
CANOUT1[12].2 :=SlowTurnRCBX;   (* SLOWTURNING RC*)
CANOUT1[12].3 :=AHEAD;(* AHEAD*)
CANOUT1[12].4 :=ASTERN;  (*ASTERN*)
CANOUT1[12].5 :=H_AIRRUN_BR_ECR;(*AIRRUN_RC_BX;   AIR RUN RC*)
CANOUT1[12].6 :=SlowTurnFailResetRC;   (*SLOWTURNING FAILURE RESET RC*)
CANOUT1[12].7 :=AuxBlowerPreselectedRC;(*AUX.BLOWER PRESELECT RC*)

CANOUT1[13].0 :=SPEED_PRGM_OVERD_BX;   (*SPEED PROGRAM OVERRIDE 0061*)
CANOUT1[13].1 :=CANCEL_LIMITS_BX;(* RC CANCEL LIMITS 0062*)
CANOUT1[13].2  :=  SHAFT_GENERATOR_BREAKER;(* SHAFT GENERATOR ENGAGED 0063 *)


(*CANOUT[14]   CANOUT[15]  CONTROL TRANSFER COMMANDS   0X2004  *)
CANOUT1[14].0 :=BR_PUS_SGNL_BR_CTRL;(*BRIDGE PUSHBUTTON  "BRIDGE CONTROL"0014*)
CANOUT1[14].1 :=BR_PUS_SGNL_ECRA_CTRL ;(*BRIDGE PUSHBUTTON  "MCR AUTOM. CONTROL"  0016*)
CANOUT1[14].2 :=BR_PUS_SGNL_ECRM_CTRL;  (*BRIDGE PUSHBUTTON  "MCR MAN. CONTROL"0018*)
CANOUT1[14].3 :=BR_PUS_SGNL_LOC_MAN_CTRL;(*BRIDGE PUSHBUTTON  "LOCAL MAN. CONTROL" 0020*)
CANOUT1[14].4 := ECRA_PUS_SGNL_BR_CTRL;(*MCR AUTOM. PUSHBUTTON  "BRIDGE CONTROL"  0028*)
CANOUT1[14].5 :=ECRA_PUS_SGNL_ECRA_CTRL; (*MCR AUTOM. PUSHBUTTON  "MCR AUTOM. CONTROL" 0030*)
CANOUT1[14].6 :=0; (*ECRA_PUS_ECRM_CTRL_INPUT; (*MCR AUTOM. PUSHBUTTON  "MCR MAN. CONTROL"0032*)*)
CANOUT1[14].7 :=ECRA_PUS_SGNL_LOC_MAN_CTRL;(*MCR AUTOM. PUSHBUTTON  "LOCAL MAN. CONTROL" 0034*)

CANOUT1[15].0 :=RC_HANDLE_MATCH;(*RC HANDLE MATCH*)





(**can2******)
(*--------- CANOUT1[10]   CANOUT1[11]  for  speed setpoint-----------*)

Temp_Word:=REAL_TO_WORD(SPEED_SETPOINT_BX*10);
CANOUT2[10]:=WORD_TO_BYTE(Temp_Word);
CANOUT2[11]:=WORD_TO_BYTE(SHR(Temp_Word ,8));

(*CANOUT[12]   CANOUT[13] store ENGINE COMMANDS   0X2003  *)
CANOUT2[12].0 := STOP ;(*STOP 0022*)
CANOUT2[12].1 :=START_BRAKE;(*START BREAK 0016*)
CANOUT2[12].2 :=SlowTurnRCBX;   (* SLOWTURNING RC*)
CANOUT2[12].3 :=AHEAD;(* AHEAD*)
CANOUT2[12].4 :=ASTERN;  (*ASTERN*)
CANOUT2[12].5 :=H_AIRRUN_BR_ECR;(*AIRRUN_RC_BX;   AIR RUN RC*)
CANOUT2[12].6 :=SlowTurnFailResetRC;   (*SLOWTURNING FAILURE RESET RC*)
CANOUT2[12].7 :=AuxBlowerPreselectedRC;(*AUX.BLOWER PRESELECT RC*)

CANOUT2[13].0 :=SPEED_PRGM_OVERD_BX;   (*SPEED PROGRAM OVERRIDE 0061*)
CANOUT2[13].1 :=CANCEL_LIMITS_BX;(* RC CANCEL LIMITS 0062*)
CANOUT2[13].2  :=  SHAFT_GENERATOR_BREAKER;(* SHAFT GENERATOR ENGAGED 0063 *)

(*CANOUT[14]   CANOUT[15]  CONTROL TRANSFER COMMANDS   0X2004  *)
CANOUT2[14].0 :=BR_PUS_SGNL_BR_CTRL;(*BRIDGE PUSHBUTTON  "BRIDGE CONTROL"0014*)
CANOUT2[14].1 :=BR_PUS_SGNL_ECRA_CTRL ;(*BRIDGE PUSHBUTTON  "MCR AUTOM. CONTROL"  0016*)
CANOUT2[14].2 :=BR_PUS_SGNL_ECRM_CTRL;  (*BRIDGE PUSHBUTTON  "MCR MAN. CONTROL"0018*)
CANOUT2[14].3 :=BR_PUS_SGNL_LOC_MAN_CTRL;(*BRIDGE PUSHBUTTON  "LOCAL MAN. CONTROL" 0020*)
CANOUT2[14].4 := ECRA_PUS_SGNL_BR_CTRL;(*MCR AUTOM. PUSHBUTTON  "BRIDGE CONTROL"  0028*)
CANOUT2[14].5 :=ECRA_PUS_SGNL_ECRA_CTRL; (*MCR AUTOM. PUSHBUTTON  "MCR AUTOM. CONTROL" 0030*)
CANOUT2[14].6 :=0; (*ECRA_PUS_ECRM_CTRL_INPUT; (*MCR AUTOM. PUSHBUTTON  "MCR MAN. CONTROL"0032*)*)
CANOUT2[14].7 :=ECRA_PUS_SGNL_LOC_MAN_CTRL;(*MCR AUTOM. PUSHBUTTON  "LOCAL MAN. CONTROL" 0034*)

CANOUT2[15].0 :=RC_HANDLE_MATCH;(*RC HANDLE MATCH*)


(***若发送的数据有变化，则立刻发送数据出去***)
(*CANOUT1,CANOUT2 数据一样，故只需判断 CANOUT1 数据是否发生变化*)
(*if  data changed, update old CAN ARRAY*)
FOR	I := 0 TO 15	DO
	IF	CANOUT1[10 + I] <> CANOUT_OLD[10 + I]
	THEN
		(*set  data  change flag  true*)
		DATA_CHANGE_CAN1 := TRUE;

		(*update old CAN ARRAY*)
		CANOUT_OLD[10 + I] := CANOUT1[10 + I];
	END_IF
END_FOR


(* if   data changed  , then  send date group1 out  immediately *)
IF	DATA_CHANGE_CAN1 = TRUE
THEN
	CANOUT1[6].0 := NOT  CANOUT1[6].0;
	CANOUT2[6].0 := NOT  CANOUT2[6].0;

	DATA_CHANGE_CAN1 := FALSE;
END_IF
END_FUNCTION_BLOCK

(* POU SPEED_MEASUREMENT_RCS, LD *)
PROGRAM SPEED_MEASUREMENT_RCS

VAR
	Position_Low: DINT;
	Position_High: DINT;
	Position_Last_Cycle_1000MS: DINT;
	Position_Last_Cycle_50MS: DINT;
	TURNING_AHEAD_RCS_NPN: BOOL;
	TURNING_ASTERN_RCS_NPN: BOOL;
	Position: DINT;
	STANDSTILL_RCS_NPN: BOOL;
	COUNT_DIFF_1000MS: DINT;
	TEETH_COUNTER_FOR_STANDSTILL_LIMIT_PER_MIN: INT;
	TEETH_COUNTER_FOR_STANDSTILL_LIMIT_PER_SEC: INT;
	OUT_OF_STANDSTILL_LIMIT: BOOL;
	BLINK1: BLINK;
	RT1: R_TRIG;
	ACTIVE_1000MS: BOOL;
	temp1: INT;
	temp2: DINT;
	temp3: INT;
	temp_no_use:BOOL;
	STANDSTILL_RCS_ANALOG: BOOL;
	DIAG1: GET_TERMINALDIAG;
	T1: TON;
	BLINK2: BLINK;
	RT2: R_TRIG;
	RT123: R_TRIG;
	ACTIVE_50MS: BOOL;
	TEETH_COUNTER_FOR_OVERSPEED_LIMIT_PER_50MS: INT;
	TEETH_COUNTER_FOR_OVERSPEED_LIMIT_PER_MIN: INT;
	COUNT_DIFF_50MS: DINT;
	Position_for_revolution_counter: DINT;
	COUNT_DIFF_revolution_counter: DINT;
	TEETH_PER_COUNT_FOR_REVOLUTION_COUNTER: INT;
	REACH_ONE_COUNT: BOOL;
	RT3: R_TRIG;
	ANALOG_DETECT_SPEED_M:REAL;(* INT;*)
	COUNT_DIFF_1000MS_ZERO: BOOL;
	T3: TOF;
	T4: TOF;
	COUNT_DECLINE: BOOL;
	COUNT_DIFF_1000MS_ABS: DINT;
	TURNING_ASTERN_RCS_NPN_M: BOOL;
	NPN_DETECT_SPEED_RCS_M: INT;
	RAMP1: RAMP_REAL;
	OVERSPEED_RCS_TEMP_M: BOOL;
	OVERSPEED_RCS_TEMP_M_M1: BOOL;
	OVERSPEED_RCS_TEMP_M_M2:BOOL;
	OVERSPEED_RCS_SIMULATION: BOOL;
	RCS_SPEED_MEANSURE_VALUE_INT: INT;
END_VAR
VAR_INPUT

	STANDSTILL_ESS: BOOL; (* From ESS through Modbus.Note: Need to be added in the communication between RCS and ESS *)
	TURNING_AHEAD_ESS: BOOL; (* From ESS through Modbus *)
	TURNING_ASTERN_ESS: BOOL; (* From ESS through Modbus *)
	(*GEAR_TEETH_PER_REVOLUTION_SETPOINT: INT;  Setpoint from HMI  move to GLOBAL_VAR*)
	(* STANDSTILL_SETPOINT: INT; Setpoint from HMI  move to GLOBAL_VAR*)
	(* OVERSPEED_SETPOINT: INT;  Setpoint from HMI  move to GLOBAL_VAR*)
	(* REVOLUTION_COUNTER_FACTOR_SETPOINT: INT; Setpoint from HMI  move to GLOBAL_VAR *)
END_VAR
VAR_OUTPUT
	RCS_NPN_SENSER_FAILURE: BOOL; (* Health of the RCS NPN speed dectors *)
	RCS_ANALOG_SPEED_SENSER_FAILURE: BOOL; (* Health of the RCS analog speed dector *)
	STANDSTILL_RCS: BOOL;
	TURNING_ASTERN_RCS: BOOL;
	TURNING_AHEAD_RCS: BOOL;
	 SPEED_RCS:REAL; (*INT;(*SPEED MEASURE VALUE--------------------------*)*)


END_VAR
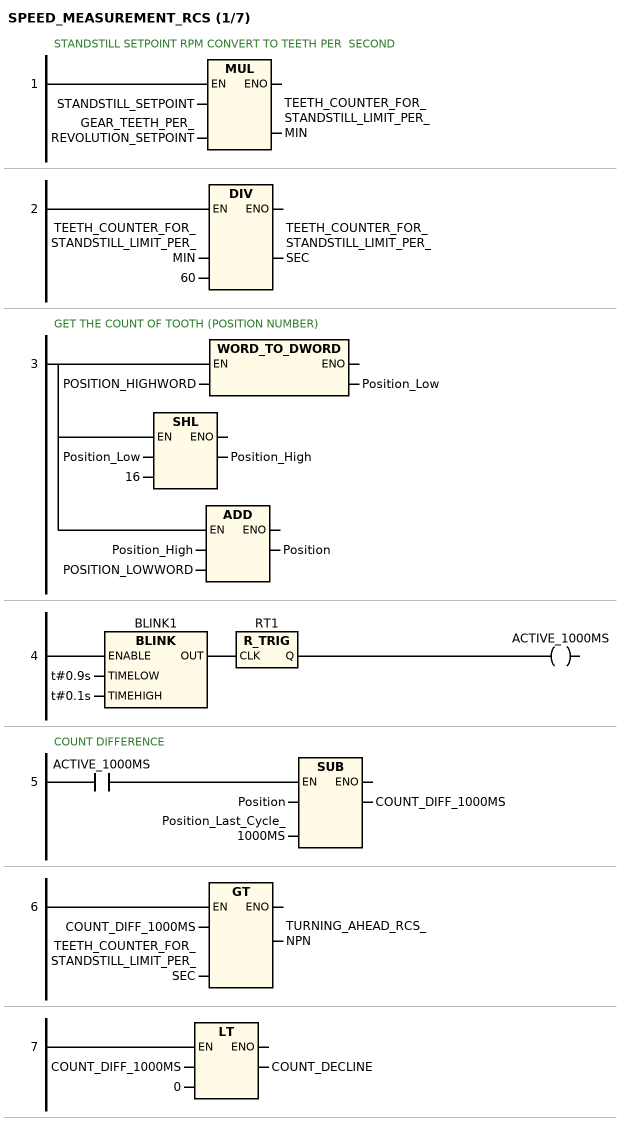
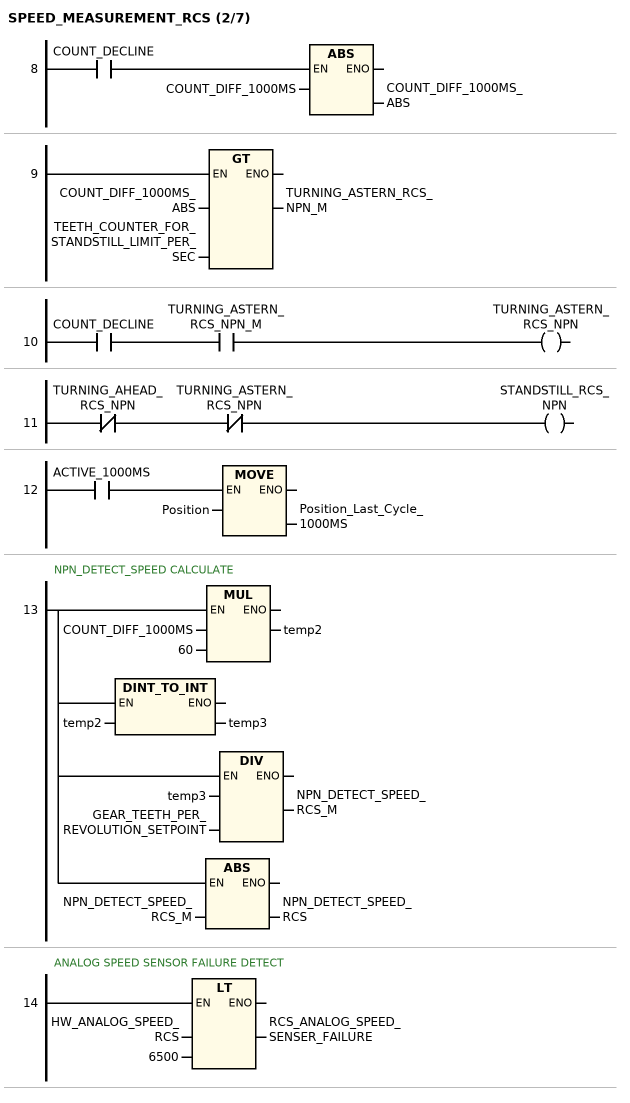
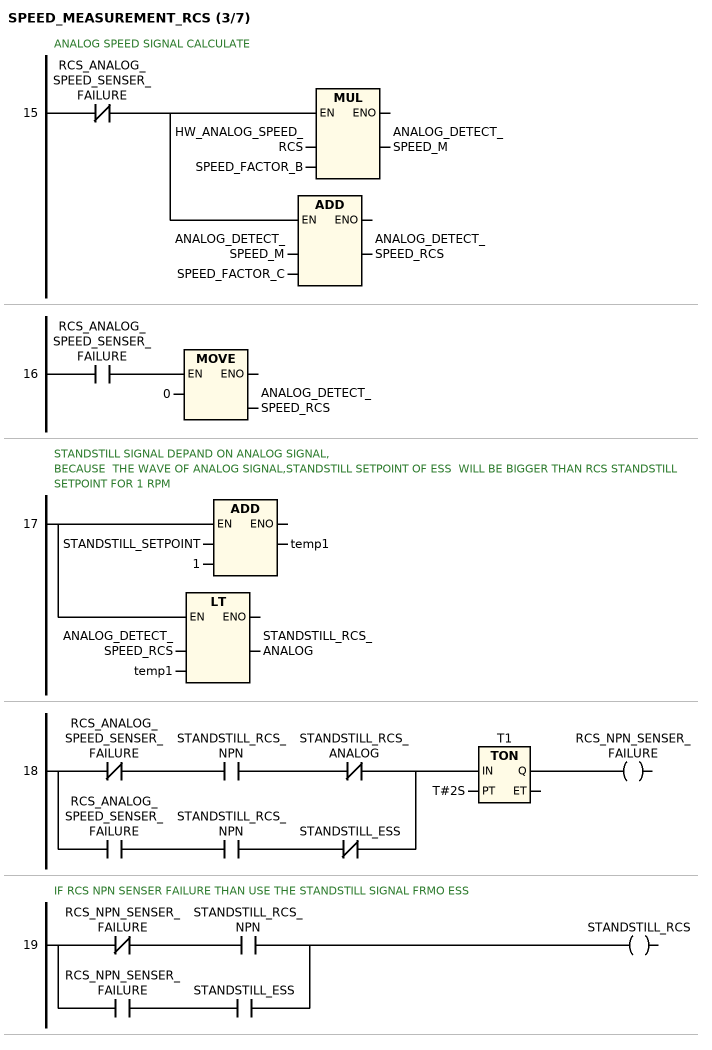
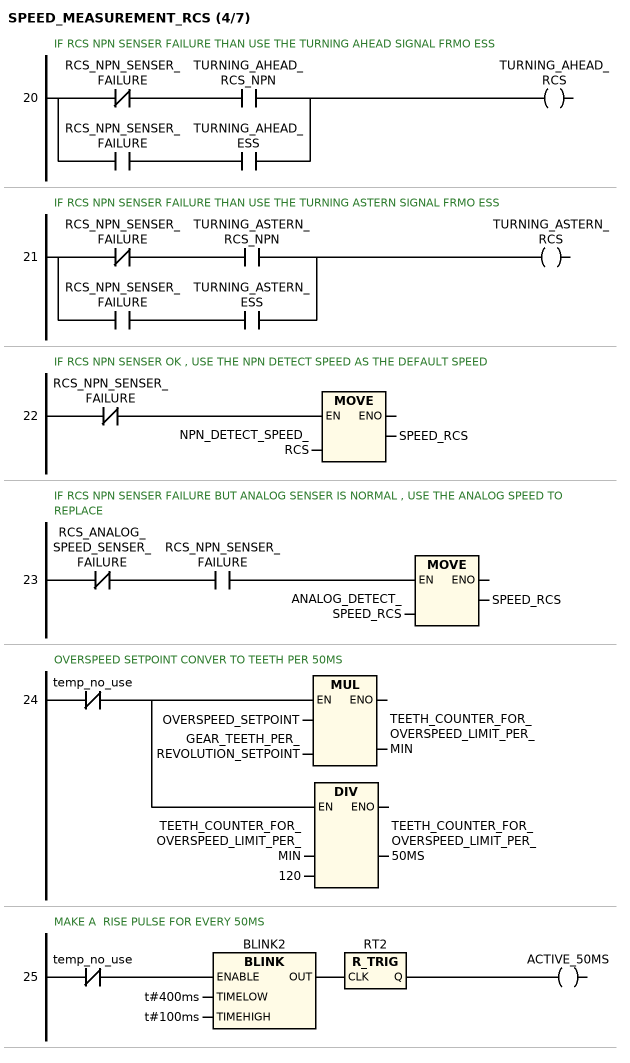
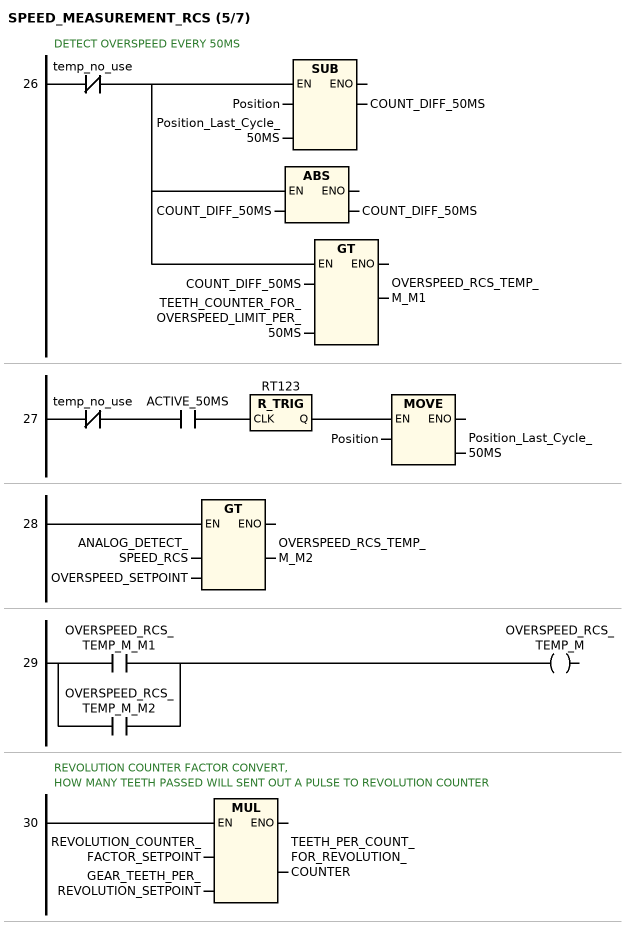
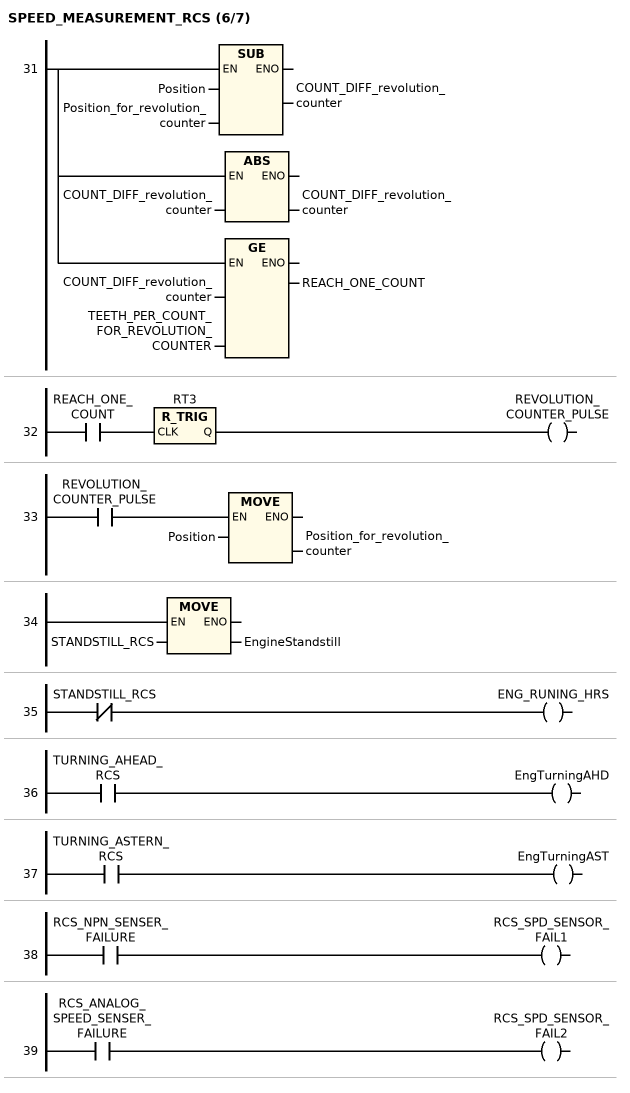
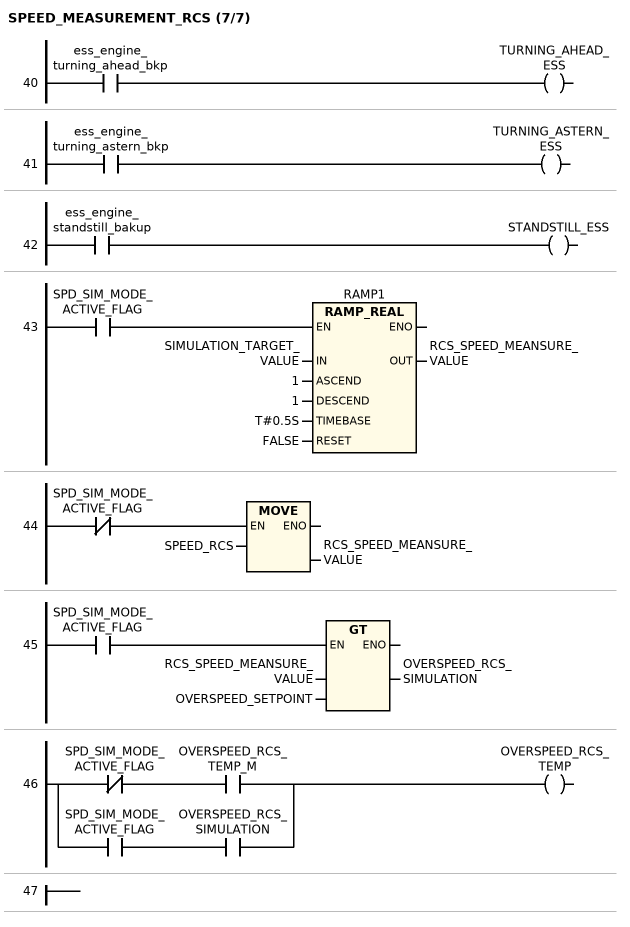
_LD_ (* Ladder Diagram *)
NETWORK 1 (* STANDSTILL SETPOINT RPM CONVERT TO TEETH PER  SECOND *)
	*
		EN --- MUL(STANDSTILL_SETPOINT, GEAR_TEETH_PER_REVOLUTION_SETPOINT) => TEETH_COUNTER_FOR_STANDSTILL_LIMIT_PER_MIN
NETWORK 2
	*
		EN --- DIV(TEETH_COUNTER_FOR_STANDSTILL_LIMIT_PER_MIN, 60) => TEETH_COUNTER_FOR_STANDSTILL_LIMIT_PER_SEC
NETWORK 3 (* GET THE COUNT OF TOOTH (POSITION NUMBER) *)
	*
		EN --- WORD_TO_DWORD(POSITION_HIGHWORD) => Position_Low
		EN --- SHL(Position_Low, 16) => Position_High
		EN --- ADD(Position_High, POSITION_LOWWORD) => Position
NETWORK 4
	BLINK1:BLINK(ENABLE: *, TIMELOW: t#0.9s, TIMEHIGH: t#0.1s) - RT1:R_TRIG(CLK: *) --- (ACTIVE_1000MS)
NETWORK 5 (* COUNT DIFFERENCE *)
	[ACTIVE_1000MS]
		EN --- SUB(Position, Position_Last_Cycle_1000MS) => COUNT_DIFF_1000MS
NETWORK 6
	*
		EN --- GT(COUNT_DIFF_1000MS, TEETH_COUNTER_FOR_STANDSTILL_LIMIT_PER_SEC) => TURNING_AHEAD_RCS_NPN
NETWORK 7
	*
		EN --- LT(COUNT_DIFF_1000MS, 0) => COUNT_DECLINE
NETWORK 8
	[COUNT_DECLINE]
		EN --- ABS(COUNT_DIFF_1000MS) => COUNT_DIFF_1000MS_ABS
NETWORK 9
	*
		EN --- GT(COUNT_DIFF_1000MS_ABS, TEETH_COUNTER_FOR_STANDSTILL_LIMIT_PER_SEC) => TURNING_ASTERN_RCS_NPN_M
NETWORK 10
	[COUNT_DECLINE] - [TURNING_ASTERN_RCS_NPN_M] --- (TURNING_ASTERN_RCS_NPN)
NETWORK 11
	[/TURNING_AHEAD_RCS_NPN] - [/TURNING_ASTERN_RCS_NPN] --- (STANDSTILL_RCS_NPN)
NETWORK 12
	[ACTIVE_1000MS]
		EN --- MOVE(Position) => Position_Last_Cycle_1000MS
NETWORK 13 (* NPN_DETECT_SPEED CALCULATE *)
	*
		EN --- MUL(COUNT_DIFF_1000MS, 60) => temp2
		EN --- DINT_TO_INT(temp2) => temp3
		EN --- DIV(temp3, GEAR_TEETH_PER_REVOLUTION_SETPOINT) => NPN_DETECT_SPEED_RCS_M
		EN --- ABS(NPN_DETECT_SPEED_RCS_M) => NPN_DETECT_SPEED_RCS
NETWORK 14 (* ANALOG SPEED SENSOR FAILURE DETECT *)
	*
		EN --- LT(HW_ANALOG_SPEED_RCS, 6500) => RCS_ANALOG_SPEED_SENSER_FAILURE
NETWORK 15 (* ANALOG SPEED SIGNAL CALCULATE *)
	[/RCS_ANALOG_SPEED_SENSER_FAILURE]
		EN --- MUL(HW_ANALOG_SPEED_RCS, SPEED_FACTOR_B) => ANALOG_DETECT_SPEED_M
		EN --- ADD(ANALOG_DETECT_SPEED_M, SPEED_FACTOR_C) => ANALOG_DETECT_SPEED_RCS
NETWORK 16
	[RCS_ANALOG_SPEED_SENSER_FAILURE]
		EN --- MOVE(0) => ANALOG_DETECT_SPEED_RCS
NETWORK 17 (* STANDSTILL SIGNAL DEPAND ON ANALOG SIGNAL, / BECAUSE  THE WAVE OF ANALOG SIGNAL,STANDSTILL SETPOINT OF ESS  WILL BE BIGGER THAN RCS STANDSTILL SETPOINT FOR 1 RPM *)
	*
		EN --- ADD(STANDSTILL_SETPOINT, 1) => temp1
		EN --- LT(ANALOG_DETECT_SPEED_RCS, temp1) => STANDSTILL_RCS_ANALOG
NETWORK 18
	{ [/RCS_ANALOG_SPEED_SENSER_FAILURE] - [STANDSTILL_RCS_NPN] - [/STANDSTILL_RCS_ANALOG] | [RCS_ANALOG_SPEED_SENSER_FAILURE] - [STANDSTILL_RCS_NPN] - [/STANDSTILL_ESS] } - T1:TON(IN: *, PT: T#2S) --- (RCS_NPN_SENSER_FAILURE)
NETWORK 19 (* IF RCS NPN SENSER FAILURE THAN USE THE STANDSTILL SIGNAL FRMO ESS *)
	{ [/RCS_NPN_SENSER_FAILURE] - [STANDSTILL_RCS_NPN] | [RCS_NPN_SENSER_FAILURE] - [STANDSTILL_ESS] } --- (STANDSTILL_RCS)
NETWORK 20 (* IF RCS NPN SENSER FAILURE THAN USE THE TURNING AHEAD SIGNAL FRMO ESS *)
	{ [/RCS_NPN_SENSER_FAILURE] - [TURNING_AHEAD_RCS_NPN] | [RCS_NPN_SENSER_FAILURE] - [TURNING_AHEAD_ESS] } --- (TURNING_AHEAD_RCS)
NETWORK 21 (* IF RCS NPN SENSER FAILURE THAN USE THE TURNING ASTERN SIGNAL FRMO ESS *)
	{ [/RCS_NPN_SENSER_FAILURE] - [TURNING_ASTERN_RCS_NPN] | [RCS_NPN_SENSER_FAILURE] - [TURNING_ASTERN_ESS] } --- (TURNING_ASTERN_RCS)
NETWORK 22 (* IF RCS NPN SENSER OK , USE THE NPN DETECT SPEED AS THE DEFAULT SPEED *)
	[/RCS_NPN_SENSER_FAILURE]
		EN --- MOVE(NPN_DETECT_SPEED_RCS) => SPEED_RCS
NETWORK 23 (* IF RCS NPN SENSER FAILURE BUT ANALOG SENSER IS NORMAL , USE THE ANALOG SPEED TO REPLACE *)
	[/RCS_ANALOG_SPEED_SENSER_FAILURE] - [RCS_NPN_SENSER_FAILURE]
		EN --- MOVE(ANALOG_DETECT_SPEED_RCS) => SPEED_RCS
NETWORK 24 (* OVERSPEED SETPOINT CONVER TO TEETH PER 50MS *)
	[/temp_no_use]
		EN --- MUL(OVERSPEED_SETPOINT, GEAR_TEETH_PER_REVOLUTION_SETPOINT) => TEETH_COUNTER_FOR_OVERSPEED_LIMIT_PER_MIN
		EN --- DIV(TEETH_COUNTER_FOR_OVERSPEED_LIMIT_PER_MIN, 120) => TEETH_COUNTER_FOR_OVERSPEED_LIMIT_PER_50MS
NETWORK 25 (* MAKE A  RISE PULSE FOR EVERY 50MS *)
	[/temp_no_use] - BLINK2:BLINK(ENABLE: *, TIMELOW: t#400ms, TIMEHIGH: t#100ms) - RT2:R_TRIG(CLK: *) --- (ACTIVE_50MS)
NETWORK 26 (* DETECT OVERSPEED EVERY 50MS *)
	[/temp_no_use]
		EN --- SUB(Position, Position_Last_Cycle_50MS) => COUNT_DIFF_50MS
		EN --- ABS(COUNT_DIFF_50MS) => COUNT_DIFF_50MS
		EN --- GT(COUNT_DIFF_50MS, TEETH_COUNTER_FOR_OVERSPEED_LIMIT_PER_50MS) => OVERSPEED_RCS_TEMP_M_M1
NETWORK 27
	[/temp_no_use] - [ACTIVE_50MS] - RT123:R_TRIG(CLK: *)
		EN --- MOVE(Position) => Position_Last_Cycle_50MS
NETWORK 28
	*
		EN --- GT(ANALOG_DETECT_SPEED_RCS, OVERSPEED_SETPOINT) => OVERSPEED_RCS_TEMP_M_M2
NETWORK 29
	{ [OVERSPEED_RCS_TEMP_M_M1] | [OVERSPEED_RCS_TEMP_M_M2] } --- (OVERSPEED_RCS_TEMP_M)
NETWORK 30 (* REVOLUTION COUNTER FACTOR CONVERT, / HOW MANY TEETH PASSED WILL SENT OUT A PULSE TO REVOLUTION COUNTER *)
	*
		EN --- MUL(REVOLUTION_COUNTER_FACTOR_SETPOINT, GEAR_TEETH_PER_REVOLUTION_SETPOINT) => TEETH_PER_COUNT_FOR_REVOLUTION_COUNTER
NETWORK 31
	*
		EN --- SUB(Position, Position_for_revolution_counter) => COUNT_DIFF_revolution_counter
		EN --- ABS(COUNT_DIFF_revolution_counter) => COUNT_DIFF_revolution_counter
		EN --- GE(COUNT_DIFF_revolution_counter, TEETH_PER_COUNT_FOR_REVOLUTION_COUNTER) => REACH_ONE_COUNT
NETWORK 32
	[REACH_ONE_COUNT] - RT3:R_TRIG(CLK: *) --- (REVOLUTION_COUNTER_PULSE)
NETWORK 33
	[REVOLUTION_COUNTER_PULSE]
		EN --- MOVE(Position) => Position_for_revolution_counter
NETWORK 34
	*
		EN --- MOVE(STANDSTILL_RCS) => EngineStandstill
NETWORK 35
	[/STANDSTILL_RCS] --- (ENG_RUNING_HRS)
NETWORK 36
	[TURNING_AHEAD_RCS] --- (EngTurningAHD)
NETWORK 37
	[TURNING_ASTERN_RCS] --- (EngTurningAST)
NETWORK 38
	[RCS_NPN_SENSER_FAILURE] --- (RCS_SPD_SENSOR_FAIL1)
NETWORK 39
	[RCS_ANALOG_SPEED_SENSER_FAILURE] --- (RCS_SPD_SENSOR_FAIL2)
NETWORK 40
	[ess_engine_turning_ahead_bkp] --- (TURNING_AHEAD_ESS)
NETWORK 41
	[ess_engine_turning_astern_bkp] --- (TURNING_ASTERN_ESS)
NETWORK 42
	[ess_engine_standstill_bakup] --- (STANDSTILL_ESS)
NETWORK 43
	[SPD_SIM_MODE_ACTIVE_FLAG]
		EN --- RAMP1:RAMP_REAL(IN: SIMULATION_TARGET_VALUE, ASCEND: 1, DESCEND: 1, TIMEBASE: T#0.5S, RESET: FALSE) => RCS_SPEED_MEANSURE_VALUE
NETWORK 44
	[/SPD_SIM_MODE_ACTIVE_FLAG]
		EN --- MOVE(SPEED_RCS) => RCS_SPEED_MEANSURE_VALUE
NETWORK 45
	[SPD_SIM_MODE_ACTIVE_FLAG]
		EN --- GT(RCS_SPEED_MEANSURE_VALUE, OVERSPEED_SETPOINT) => OVERSPEED_RCS_SIMULATION
NETWORK 46
	{ [/SPD_SIM_MODE_ACTIVE_FLAG] - [OVERSPEED_RCS_TEMP_M] | [SPD_SIM_MODE_ACTIVE_FLAG] - [OVERSPEED_RCS_SIMULATION] } --- (OVERSPEED_RCS_TEMP)
NETWORK 47
	*
_END_LD_
(* the same logic as Structured Text *)
(* Network 1: STANDSTILL SETPOINT RPM CONVERT TO TEETH PER  SECOND *)
TEETH_COUNTER_FOR_STANDSTILL_LIMIT_PER_MIN := STANDSTILL_SETPOINT * GEAR_TEETH_PER_REVOLUTION_SETPOINT;
(* Network 2 *)
TEETH_COUNTER_FOR_STANDSTILL_LIMIT_PER_SEC := TEETH_COUNTER_FOR_STANDSTILL_LIMIT_PER_MIN / 60;
(* Network 3: GET THE COUNT OF TOOTH (POSITION NUMBER) *)
Position_Low := WORD_TO_DWORD(POSITION_HIGHWORD);
Position_High := SHL(Position_Low, 16);
Position := Position_High + POSITION_LOWWORD;
(* Network 4 *)
BLINK1(ENABLE := TRUE, TIMELOW := t#0.9s, TIMEHIGH := t#0.1s);
RT1(CLK := BLINK1.OUT);
ACTIVE_1000MS := RT1.Q;
(* Network 5: COUNT DIFFERENCE *)
IF ACTIVE_1000MS THEN
	COUNT_DIFF_1000MS := Position - Position_Last_Cycle_1000MS;
END_IF;
(* Network 6 *)
TURNING_AHEAD_RCS_NPN := COUNT_DIFF_1000MS > TEETH_COUNTER_FOR_STANDSTILL_LIMIT_PER_SEC;
(* Network 7 *)
COUNT_DECLINE := COUNT_DIFF_1000MS < 0;
(* Network 8 *)
IF COUNT_DECLINE THEN
	COUNT_DIFF_1000MS_ABS := ABS(COUNT_DIFF_1000MS);
END_IF;
(* Network 9 *)
TURNING_ASTERN_RCS_NPN_M := COUNT_DIFF_1000MS_ABS > TEETH_COUNTER_FOR_STANDSTILL_LIMIT_PER_SEC;
(* Network 10 *)
TURNING_ASTERN_RCS_NPN := COUNT_DECLINE AND TURNING_ASTERN_RCS_NPN_M;
(* Network 11 *)
STANDSTILL_RCS_NPN := NOT TURNING_AHEAD_RCS_NPN AND NOT TURNING_ASTERN_RCS_NPN;
(* Network 12 *)
IF ACTIVE_1000MS THEN
	Position_Last_Cycle_1000MS := Position;
END_IF;
(* Network 13: NPN_DETECT_SPEED CALCULATE *)
temp2 := COUNT_DIFF_1000MS * 60;
temp3 := DINT_TO_INT(temp2);
NPN_DETECT_SPEED_RCS_M := temp3 / GEAR_TEETH_PER_REVOLUTION_SETPOINT;
NPN_DETECT_SPEED_RCS := ABS(NPN_DETECT_SPEED_RCS_M);
(* Network 14: ANALOG SPEED SENSOR FAILURE DETECT *)
RCS_ANALOG_SPEED_SENSER_FAILURE := HW_ANALOG_SPEED_RCS < 6500;
(* Network 15: ANALOG SPEED SIGNAL CALCULATE *)
IF NOT RCS_ANALOG_SPEED_SENSER_FAILURE THEN
	ANALOG_DETECT_SPEED_M := HW_ANALOG_SPEED_RCS * SPEED_FACTOR_B;
	ANALOG_DETECT_SPEED_RCS := ANALOG_DETECT_SPEED_M + SPEED_FACTOR_C;
END_IF;
(* Network 16 *)
IF RCS_ANALOG_SPEED_SENSER_FAILURE THEN
	ANALOG_DETECT_SPEED_RCS := 0;
END_IF;
(* Network 17: STANDSTILL SIGNAL DEPAND ON ANALOG SIGNAL, / BECAUSE  THE WAVE OF ANALOG SIGNAL,STANDSTILL SETPOINT OF ESS  WILL BE BIGGER THAN RCS STANDSTILL SETPOINT FOR 1 RPM *)
temp1 := STANDSTILL_SETPOINT + 1;
STANDSTILL_RCS_ANALOG := ANALOG_DETECT_SPEED_RCS < temp1;
(* Network 18 *)
T1(IN := NOT RCS_ANALOG_SPEED_SENSER_FAILURE AND STANDSTILL_RCS_NPN AND NOT STANDSTILL_RCS_ANALOG OR RCS_ANALOG_SPEED_SENSER_FAILURE AND STANDSTILL_RCS_NPN AND NOT STANDSTILL_ESS, PT := T#2S);
RCS_NPN_SENSER_FAILURE := T1.Q;
(* Network 19: IF RCS NPN SENSER FAILURE THAN USE THE STANDSTILL SIGNAL FRMO ESS *)
STANDSTILL_RCS := NOT RCS_NPN_SENSER_FAILURE AND STANDSTILL_RCS_NPN OR RCS_NPN_SENSER_FAILURE AND STANDSTILL_ESS;
(* Network 20: IF RCS NPN SENSER FAILURE THAN USE THE TURNING AHEAD SIGNAL FRMO ESS *)
TURNING_AHEAD_RCS := NOT RCS_NPN_SENSER_FAILURE AND TURNING_AHEAD_RCS_NPN OR RCS_NPN_SENSER_FAILURE AND TURNING_AHEAD_ESS;
(* Network 21: IF RCS NPN SENSER FAILURE THAN USE THE TURNING ASTERN SIGNAL FRMO ESS *)
TURNING_ASTERN_RCS := NOT RCS_NPN_SENSER_FAILURE AND TURNING_ASTERN_RCS_NPN OR RCS_NPN_SENSER_FAILURE AND TURNING_ASTERN_ESS;
(* Network 22: IF RCS NPN SENSER OK , USE THE NPN DETECT SPEED AS THE DEFAULT SPEED *)
IF NOT RCS_NPN_SENSER_FAILURE THEN
	SPEED_RCS := NPN_DETECT_SPEED_RCS;
END_IF;
(* Network 23: IF RCS NPN SENSER FAILURE BUT ANALOG SENSER IS NORMAL , USE THE ANALOG SPEED TO REPLACE *)
IF NOT RCS_ANALOG_SPEED_SENSER_FAILURE AND RCS_NPN_SENSER_FAILURE THEN
	SPEED_RCS := ANALOG_DETECT_SPEED_RCS;
END_IF;
(* Network 24: OVERSPEED SETPOINT CONVER TO TEETH PER 50MS *)
IF NOT temp_no_use THEN
	TEETH_COUNTER_FOR_OVERSPEED_LIMIT_PER_MIN := OVERSPEED_SETPOINT * GEAR_TEETH_PER_REVOLUTION_SETPOINT;
	TEETH_COUNTER_FOR_OVERSPEED_LIMIT_PER_50MS := TEETH_COUNTER_FOR_OVERSPEED_LIMIT_PER_MIN / 120;
END_IF;
(* Network 25: MAKE A  RISE PULSE FOR EVERY 50MS *)
BLINK2(ENABLE := NOT temp_no_use, TIMELOW := t#400ms, TIMEHIGH := t#100ms);
RT2(CLK := BLINK2.OUT);
ACTIVE_50MS := RT2.Q;
(* Network 26: DETECT OVERSPEED EVERY 50MS *)
IF NOT temp_no_use THEN
	COUNT_DIFF_50MS := Position - Position_Last_Cycle_50MS;
	COUNT_DIFF_50MS := ABS(COUNT_DIFF_50MS);
	OVERSPEED_RCS_TEMP_M_M1 := COUNT_DIFF_50MS > TEETH_COUNTER_FOR_OVERSPEED_LIMIT_PER_50MS;
END_IF;
(* Network 27 *)
RT123(CLK := NOT temp_no_use AND ACTIVE_50MS);
IF RT123.Q THEN
	Position_Last_Cycle_50MS := Position;
END_IF;
(* Network 28 *)
OVERSPEED_RCS_TEMP_M_M2 := ANALOG_DETECT_SPEED_RCS > OVERSPEED_SETPOINT;
(* Network 29 *)
OVERSPEED_RCS_TEMP_M := OVERSPEED_RCS_TEMP_M_M1 OR OVERSPEED_RCS_TEMP_M_M2;
(* Network 30: REVOLUTION COUNTER FACTOR CONVERT, / HOW MANY TEETH PASSED WILL SENT OUT A PULSE TO REVOLUTION COUNTER *)
TEETH_PER_COUNT_FOR_REVOLUTION_COUNTER := REVOLUTION_COUNTER_FACTOR_SETPOINT * GEAR_TEETH_PER_REVOLUTION_SETPOINT;
(* Network 31 *)
COUNT_DIFF_revolution_counter := Position - Position_for_revolution_counter;
COUNT_DIFF_revolution_counter := ABS(COUNT_DIFF_revolution_counter);
REACH_ONE_COUNT := COUNT_DIFF_revolution_counter >= TEETH_PER_COUNT_FOR_REVOLUTION_COUNTER;
(* Network 32 *)
RT3(CLK := REACH_ONE_COUNT);
REVOLUTION_COUNTER_PULSE := RT3.Q;
(* Network 33 *)
IF REVOLUTION_COUNTER_PULSE THEN
	Position_for_revolution_counter := Position;
END_IF;
(* Network 34 *)
EngineStandstill := STANDSTILL_RCS;
(* Network 35 *)
ENG_RUNING_HRS := NOT STANDSTILL_RCS;
(* Network 36 *)
EngTurningAHD := TURNING_AHEAD_RCS;
(* Network 37 *)
EngTurningAST := TURNING_ASTERN_RCS;
(* Network 38 *)
RCS_SPD_SENSOR_FAIL1 := RCS_NPN_SENSER_FAILURE;
(* Network 39 *)
RCS_SPD_SENSOR_FAIL2 := RCS_ANALOG_SPEED_SENSER_FAILURE;
(* Network 40 *)
TURNING_AHEAD_ESS := ess_engine_turning_ahead_bkp;
(* Network 41 *)
TURNING_ASTERN_ESS := ess_engine_turning_astern_bkp;
(* Network 42 *)
STANDSTILL_ESS := ess_engine_standstill_bakup;
(* Network 43 *)
IF SPD_SIM_MODE_ACTIVE_FLAG THEN
	RAMP1(IN := SIMULATION_TARGET_VALUE, ASCEND := 1, DESCEND := 1, TIMEBASE := T#0.5S, RESET := FALSE);
	RCS_SPEED_MEANSURE_VALUE := RAMP1.OUT;
END_IF;
(* Network 44 *)
IF NOT SPD_SIM_MODE_ACTIVE_FLAG THEN
	RCS_SPEED_MEANSURE_VALUE := SPEED_RCS;
END_IF;
(* Network 45 *)
IF SPD_SIM_MODE_ACTIVE_FLAG THEN
	OVERSPEED_RCS_SIMULATION := RCS_SPEED_MEANSURE_VALUE > OVERSPEED_SETPOINT;
END_IF;
(* Network 46 *)
OVERSPEED_RCS_TEMP := NOT SPD_SIM_MODE_ACTIVE_FLAG AND OVERSPEED_RCS_TEMP_M OR SPD_SIM_MODE_ACTIVE_FLAG AND OVERSPEED_RCS_SIMULATION;
(* Network 47 *)
END_PROGRAM

(* POU HeartBeat_Receive, ST *)
PROGRAM HeartBeat_Receive
VAR
	HeartBeatBit: BOOL;
	CAN1:CAN_Communication;
	CAN2:CAN_Communication;

	reset1: BOOL;
	reset2: BOOL;
	size: BYTE;
	IN1 AT %IB0 : ARRAY[0..47] OF BYTE;
	OUT1 AT %QB0 : ARRAY[0..47] OF BYTE;

	IN2 AT %IB48 : ARRAY[0..47] OF BYTE;
	OUT2 AT %QB48 : ARRAY[0..47] OF BYTE;

	eStatus: CAN_eStatus;
	mdata1: POINTER TO MBX_typDataConfig;
	wCOBID1: WORD;
	ENABLE: BOOL;
	wCOBID2: WORD;


	(*CAN1 , CAN2 time out  TIMER*)
	CAN1_TIMEOUT_TIMER: TON;
	CAN2_TIMEOUT_TIMER: TON;



END_VAR
(*HeartBeat from UNIC         *)
CAN1(	xEnable:=TRUE ,ptInModule:=ADR(CANIN1) ,ptOutModule:=ADR(OUT1) ,bSizeAcyclicChannel:=5 ,bSizeModule750_658:=48 ,xResetAcyclicChannel:=reset1 ,
	      xResetCANChannel:=reset2 ,bActualSizeModule750_658=>size ,eStatus=>eStatus ,	xAcyclicChannelError=> ,eAcyclicChannelError=> ,xCanChannelError=> ,eCanChannelError=> );
CAN2(	xEnable:=TRUE ,ptInModule:=ADR(CANIN2) ,ptOutModule:=ADR(OUT2) ,bSizeAcyclicChannel:=5 ,bSizeModule750_658:=48 ,xResetAcyclicChannel:=reset1 ,
	      xResetCANChannel:=reset2 ,bActualSizeModule750_658=>size ,eStatus=>eStatus ,	xAcyclicChannelError=> ,eAcyclicChannelError=> ,xCanChannelError=> ,eCanChannelError=> );

(*---------------------CAN1---------------------*)
IF CANIN1_CHG_FLAG THEN

	CAN1_TIMEOUT_TIMER(IN := FALSE);
END_IF
wCOBID1:=IN1[3]*8+IN1[4]/32;
IF IN1[5]=5  AND wCOBID1=16#711 THEN
	(*STGP TIMER*)
	CAN1_TIMEOUT_TIMER(IN := FALSE);
      BreakDownCAN1:=FALSE;
ELSE
	(*if there is not received HeartBeat frame,then start timeout  timer,  3s time out*)
	CAN1_TIMEOUT_TIMER(IN := TRUE, PT := t#3s);
END_IF

IF  CAN1_TIMEOUT_TIMER.Q = TRUE(*it will  change  CAN  when  didn't  receive HBeat  more than 3s (or three times) *)
THEN
             BreakDownCAN1:=TRUE;
END_IF
(*%QX48.0:=  NOT BreakDownCAN1;*)


(*--------------------CAN2--------------------*)
IF CANIN2_CHG_FLAG THEN

	CAN2_TIMEOUT_TIMER(IN := FALSE);
END_IF
wCOBID2:=IN2[3]*8+IN2[4]/32;
IF IN2[5]=5  AND wCOBID2=16#711 THEN
	(*STGP TIMER*)
	CAN2_TIMEOUT_TIMER(IN := FALSE);
      BreakDownCAN2:=FALSE;
ELSE
	(*if there is not received HeartBeat frame,then start timeout  timer,  3s time out*)
	CAN2_TIMEOUT_TIMER(IN := TRUE, PT := t#3s);
END_IF

(*it will  change  CAN  when  didn't  receive HBeat  more than 3s (or three times) *)
IF  CAN2_TIMEOUT_TIMER.Q = TRUE(*it will  change  CAN  when  didn't  receive HBeat  more than 3s *)
THEN
             BreakDownCAN2:=TRUE;
END_IF

(*%QX48.1:=  NOT BreakDownCAN2;*)


(*-----------------------------CANopen BUS chosen------------------------------------------------------------*)
IF	BreakDownCAN1 = TRUE
	AND BreakDownCAN2  = TRUE(*both CAN lines are in break*)
THEN
	CommunicationLost :=TRUE;
ELSE
	CommunicationLost := FALSE;
END_IF
END_PROGRAM

(* POU HeartBeat_Send, ST *)
PROGRAM HeartBeat_Send
VAR
END_VAR
(*control CAN CARD  enable  or  disable  sent  data*)

(*if CAN bus error,  stop sending  data  group1*)
IF BreakDownCAN1 = TRUE
THEN
  	CANOUT1[6].0:= CANOUT1[6].0;
ELSE
 	CANOUT1[6].0:=NOT CANOUT1[6].0;
END_IF

IF BreakDownCAN2 = TRUE
THEN
       CANOUT2[6].0:= CANOUT2[6].0;
ELSE
 	CANOUT2[6].0:=NOT CANOUT2[6].0;
END_IF


(*sending  HEARTBEAT  to  UNIC*)
CANOUT1[7] :=Status;
CANOUT2[7] :=Status;
(*group 2*)
CANOUT1[6].1:=NOT CANOUT1[6].1;
CANOUT2[6].1:=NOT CANOUT2[6].1;
END_PROGRAM

(* POU Generated Code/Ethernet/MBCFG_EOT, ST *)
PROGRAM MBCFG_EOT(* generated by config one prg for each slave *)

VAR_INPUT

END_VAR

VAR_OUTPUT
       BR_MVL_cfg       :    WORD;       (**) 
       ECR_MVL_cfg       :    WORD;       (**) 

    (*--- system variables (read only) ----------------------------------------*)
    MBCFG_IpAddress :   STRING(11) := '192.168.1.3'; (* address of this slave *)
    MBCFG_Port      :   UINT := 502;
    MBCFG_UnitID    :   BYTE := 3;
    MBCFG_TimeOut   :   TIME := t#50ms;
    MBCFG_Error     :   MBCFG_eERROR;
    (*-------------------------------------------------------------------------*)
END_VAR

{library private}
VAR CONSTANT
    zz_VARIABLECOUNT:   INT := 2;	(* number of variables 	*)
    zz_JOBCOUNT     :   INT := 1; 	(* number of jobs		*)
END_VAR
VAR

    (*=== VARIABLE LIST ===============================================================================*)
    zz_VariableList :   ARRAY[1..zz_VARIABLECOUNT] OF MBCFG_typVARIABLE :=
    (   BitSize         := 16,
        ptVar           := 0,
        ReadJobIndex    := 1,
        ReadStartBitNo  := 0,
        WriteJobIndex   := 0,
        WriteStartBitNo := 0 ),
    (   BitSize         := 16,
        ptVar           := 0,
        ReadJobIndex    := 1,
        ReadStartBitNo  := 16,
        WriteJobIndex   := 0,
        WriteStartBitNo := 0 )

                        ;
    (*=================================================================================================*)

    (*=== JOB LIST ====================================================================================*)
    zz_JobList     :   ARRAY[1..zz_JOBCOUNT] OF MBCFG_typCOM_JOB :=
     (   Functioncode            := 3,
        ReadStartAddress        := 512,
        ReadQuantity            := 2,
        WriteStartAddress       := 0,
        WriteQuantity           := 0,
        ptReadData              := 0, 
        ptWriteData             := 0 )

                        ;
    (*=================================================================================================*)

    (*=== DATA FIELDS =================================================================================*)
     zz_DataField_1_Read       :       ARRAY[1..2] OF WORD;
	
    (*=================================================================================================*)

    (*=== MODBUS MASTER =====================================*)
    zz_MBCFG_MASTER_ETH :       MBCFG_MASTER_UDP;
    (*=======================================================*)

END_VAR
(*--- for each variable -------------------------*)
   zz_VariableList[1].ptVar := ADR(BR_MVL_cfg);
   zz_VariableList[2].ptVar := ADR(ECR_MVL_cfg);

(*-----------------------------------------------*)

(*--- for each job -----------------------------------*)
zz_JobList[1].ptReadData   := ADR(zz_DataField_1_Read);

(*----------------------------------------------------*)


(*#### START OF FIXED CODE #####################################*)
zz_MBCFG_MASTER_ETH(	strIpAddress    := MBCFG_IpAddress,
                        uiPort          := MBCFG_Port,
                        bUnitID         := MBCFG_UnitID,
                        tTimeOut        := MBCFG_TimeOut,
                        iVariableCount  := zz_VARIABLECOUNT,
                        ptVariableList  := ADR(zz_VariableList),
                        iJobCount       := zz_JOBCOUNT,
                        ptJobList       := ADR(zz_JobList),
                        eError          => MBCFG_Error
                    );
(*##############################################################*)
END_PROGRAM
